LIN {X 0,Y 192.638,Z 331.481,A -85,B 0,C 180,E1 -21988.889,E2 -21988.889} C_VEL
LIN {X 0,Y 192.591,Z 331.489,A -85,B 0,C 180,E1 -21993.187,E2 -21993.187} C_VEL
LIN {X 0,Y 192.537,Z 331.501,A -85,B 0,C 180,E1 -21998.355,E2 -21998.355} C_VEL
LIN {X 0,Y 192.482,Z 331.497,A -85,B 0,C 180,E1 -22003.096,E2 -22003.096} C_VEL
LIN {X 0,Y 192.486,Z 331.508,A -85,B 0,C 180,E1 -22006.906,E2 -22006.906} C_VEL
LIN {X 0,Y 192.597,Z 331.632,A -85,B 0,C 180,E1 -22009.624,E2 -22009.624} C_VEL
LIN {X 0,Y 193.929,Z 336.776,A -85,B 0,C 180,E1 -22012.331,E2 -22012.331} C_VEL
LIN {X 0,Y 200.85,Z 352.206,A -85,B 0,C 180,E1 -22014.229,E2 -22014.229} C_VEL
LIN {X 0,Y 205.994,Z 365.473,A -85,B 0,C 180,E1 -22015.61,E2 -22015.61} C_VEL
LIN {X 0,Y 207.555,Z 370.626,A -85,B 0,C 180,E1 -22016.057,E2 -22016.057} C_VEL
LIN {X 0,Y 209.387,Z 387.344,A -85,B 0,C 180,E1 -22016.98,E2 -22016.98} C_VEL
LIN {X 0,Y 209.345,Z 391.227,A -85,B 0,C 180,E1 -22017.123,E2 -22017.123} C_VEL
LIN {X 0,Y 208.715,Z 395.103,A -85,B 0,C 180,E1 -22017.18,E2 -22017.18} C_VEL
LIN {X 0,Y 203.389,Z 412.296,A -85,B 0,C 180,E1 -22017.059,E2 -22017.059} C_VEL
LIN {X 0,Y 202.508,Z 418.198,A -85,B 0,C 180,E1 -22017.16,E2 -22017.16} C_VEL
LIN {X 0,Y 201.25,Z 446.446,A -85,B 0,C 180,E1 -22018.177,E2 -22018.177} C_VEL
LIN {X 0,Y 199.917,Z 460.229,A -85,B 0,C 180,E1 -22019.062,E2 -22019.062} C_VEL
LIN {X 0,Y 198.125,Z 472.398,A -85,B 0,C 180,E1 -22020.226,E2 -22020.226} C_VEL
LIN {X 0,Y 195.88,Z 485.013,A -85,B 0,C 180,E1 -22021.908,E2 -22021.908} C_VEL
LIN {X 0,Y 193.499,Z 496.249,A -85,B 0,C 180,E1 -22023.873,E2 -22023.873} C_VEL
LIN {X 0,Y 191.119,Z 506.332,A -85,B 0,C 180,E1 -22026.142,E2 -22026.142} C_VEL
LIN {X 0,Y 189.005,Z 515.48,A -85,B 0,C 180,E1 -22028.746,E2 -22028.746} C_VEL
LIN {X 0,Y 187.157,Z 523.008,A -85,B 0,C 180,E1 -22031.388,E2 -22031.388} C_VEL
LIN {X 0,Y 185.383,Z 530.39,A -85,B 0,C 180,E1 -22034.613,E2 -22034.613} C_VEL
LIN {X 0,Y 184.201,Z 536.3,A -85,B 0,C 180,E1 -22037.888,E2 -22037.888} C_VEL
LIN {X 0,Y 183.5,Z 540.938,A -85,B 0,C 180,E1 -22041.189,E2 -22041.189} C_VEL
LIN {X 0,Y 183.213,Z 543.376,A -85,B 0,C 180,E1 -22043.393,E2 -22043.393} C_VEL
LIN {X 0,Y 183.047,Z 546.146,A -85,B 0,C 180,E1 -22046.616,E2 -22046.616} C_VEL
LIN {X 0,Y 183.217,Z 548.062,A -85,B 0,C 180,E1 -22050.002,E2 -22050.002} C_VEL
LIN {X 0,Y 183.079,Z 549.003,A -85,B 0,C 180,E1 -22053.551,E2 -22053.551} C_VEL
LIN {X 0,Y 183.216,Z 548.977,A -85,B 0,C 180,E1 -22056.61,E2 -22056.61} C_VEL
LIN {X 0,Y 183.532,Z 548.51,A -85,B 0,C 180,E1 -22058.812,E2 -22058.812} C_VEL
LIN {X 0,Y 184.851,Z 546.339,A -85,B 0,C 180,E1 -22063.188,E2 -22063.188} C_VEL
LIN {X 0,Y 186.461,Z 543.652,A -85,B 0,C 180,E1 -22066.422,E2 -22066.422} C_VEL
LIN {X 0,Y 188.748,Z 539.973,A -85,B 0,C 180,E1 -22069.581,E2 -22069.581} C_VEL
LIN {X 0,Y 191.549,Z 535.205,A -85,B 0,C 180,E1 -22072.661,E2 -22072.661} C_VEL
LIN {X 0,Y 195.413,Z 528.093,A -85,B 0,C 180,E1 -22076.142,E2 -22076.142} C_VEL
LIN {X 0,Y 199.258,Z 520.373,A -85,B 0,C 180,E1 -22079.012,E2 -22079.012} C_VEL
LIN {X 0,Y 203.838,Z 510.725,A -85,B 0,C 180,E1 -22081.723,E2 -22081.723} C_VEL
LIN {X 0,Y 207.989,Z 500.784,A -85,B 0,C 180,E1 -22083.887,E2 -22083.887} C_VEL
LIN {X 0,Y 211.889,Z 489.576,A -85,B 0,C 180,E1 -22085.775,E2 -22085.775} C_VEL
LIN {X 0,Y 215.214,Z 478.603,A -85,B 0,C 180,E1 -22087.168,E2 -22087.168} C_VEL
LIN {X 0,Y 218.167,Z 466.461,A -85,B 0,C 180,E1 -22088.326,E2 -22088.326} C_VEL
LIN {X 0,Y 220.337,Z 454.664,A -85,B 0,C 180,E1 -22089.122,E2 -22089.122} C_VEL
LIN {X 0,Y 221.771,Z 441.816,A -85,B 0,C 180,E1 -22089.709,E2 -22089.709} C_VEL
LIN {X 0,Y 224.212,Z 400.799,A -85,B 0,C 180,E1 -22090.951,E2 -22090.951} C_VEL
LIN {X 0,Y 221.637,Z 393.948,A -85,B 0,C 180,E1 -22091.949,E2 -22091.949} C_VEL
LIN {X 0,Y 215.367,Z 380.157,A -85,B 0,C 180,E1 -22094.421,E2 -22094.421} C_VEL
LIN {X 0,Y 208.591,Z 367.511,A -85,B 0,C 180,E1 -22097.307,E2 -22097.307} C_VEL
LIN {X 0,Y 202.439,Z 357.412,A -85,B 0,C 180,E1 -22100.202,E2 -22100.202} C_VEL
LIN {X 0,Y 198.453,Z 351.457,A -85,B 0,C 180,E1 -22102.266,E2 -22102.266} C_VEL
LIN {X 0,Y 194.893,Z 346.176,A -85,B 0,C 180,E1 -22104.287,E2 -22104.287} C_VEL
LIN {X 0,Y 191.463,Z 341.379,A -85,B 0,C 180,E1 -22106.418,E2 -22106.418} C_VEL
LIN {X 0,Y 190.355,Z 339.981,A -85,B 0,C 180,E1 -22107.143,E2 -22107.143} C_VEL
LIN {X 0,Y 186.188,Z 334.613,A -85,B 0,C 180,E1 -22110.14,E2 -22110.14} C_VEL
LIN {X 0,Y 185.92,Z 333.953,A -85,B 0,C 180,E1 -22110.567,E2 -22110.567} C_VEL
LIN {X 0,Y 185.524,Z 332.37,A -85,B 0,C 180,E1 -22112.657,E2 -22112.657} C_VEL
LIN {X 0,Y 185.583,Z 332.358,A -85,B 0,C 180,E1 -22115.382,E2 -22115.382} C_VEL
LIN {X 0,Y 185.631,Z 332.362,A -85,B 0,C 180,E1 -22121.177,E2 -22121.177} C_VEL
LIN {X 0,Y 185.671,Z 332.35,A -85,B 0,C 180,E1 -22124.636,E2 -22124.636} C_VEL
LIN {X 0,Y 185.892,Z 332.325,A -85,B 0,C 180,E1 -22129.419,E2 -22129.419} C_VEL
LIN {X 0,Y 185.944,Z 332.316,A -85,B 0,C 180,E1 -22133.49,E2 -22133.49} C_VEL
LIN {X 0,Y 186.186,Z 332.285,A -85,B 0,C 180,E1 -22137.837,E2 -22137.837} C_VEL
LIN {X 0,Y 186.399,Z 332.249,A -85,B 0,C 180,E1 -22140,E2 -22140} C_VEL
LIN {X 0,Y 185.907,Z 332.313,A -85,B 0,C 180,E1 -22144.337,E2 -22144.337} C_VEL
LIN {X 0,Y 185.981,Z 332.306,A -85,B 0,C 180,E1 -22148.694,E2 -22148.694} C_VEL
LIN {X 0,Y 185.727,Z 332.338,A -85,B 0,C 180,E1 -22153.124,E2 -22153.124} C_VEL
LIN {X 0,Y 185.69,Z 332.458,A -85,B 0,C 180,E1 -22158.755,E2 -22158.755} C_VEL
LIN {X 0,Y 186.392,Z 334.808,A -85,B 0,C 180,E1 -22159.436,E2 -22159.436} C_VEL
LIN {X 0,Y 188.203,Z 337.049,A -85,B 0,C 180,E1 -22160.779,E2 -22160.779} C_VEL
LIN {X 0,Y 190.263,Z 338.408,A -85,B 0,C 180,E1 -22162.106,E2 -22162.106} C_VEL
LIN {X 0,Y 192.016,Z 341.447,A -85,B 0,C 180,E1 -22163.313,E2 -22163.313} C_VEL
LIN {X 0,Y 194.469,Z 343.734,A -85,B 0,C 180,E1 -22164.755,E2 -22164.755} C_VEL
LIN {X 0,Y 196.792,Z 347.187,A -85,B 0,C 180,E1 -22166.117,E2 -22166.117} C_VEL
LIN {X 0,Y 198.463,Z 348.976,A -85,B 0,C 180,E1 -22167.001,E2 -22167.001} C_VEL
LIN {X 0,Y 201.253,Z 352.699,A -85,B 0,C 180,E1 -22168.446,E2 -22168.446} C_VEL
LIN {X 0,Y 206.02,Z 359.299,A -85,B 0,C 180,E1 -22170.726,E2 -22170.726} C_VEL
LIN {X 0,Y 211.19,Z 366.859,A -85,B 0,C 180,E1 -22172.976,E2 -22172.976} C_VEL
LIN {X 0,Y 216.737,Z 376.683,A -85,B 0,C 180,E1 -22175.248,E2 -22175.248} C_VEL
LIN {X 0,Y 222.914,Z 389.306,A -85,B 0,C 180,E1 -22177.608,E2 -22177.608} C_VEL
LIN {X 0,Y 224.598,Z 393.07,A -85,B 0,C 180,E1 -22178.227,E2 -22178.227} C_VEL
LIN {X 0,Y 221.905,Z 436.193,A -85,B 0,C 180,E1 -22179.548,E2 -22179.548} C_VEL
LIN {X 0,Y 220.127,Z 449.537,A -85,B 0,C 180,E1 -22180.247,E2 -22180.247} C_VEL
LIN {X 0,Y 217.847,Z 461.771,A -85,B 0,C 180,E1 -22181.227,E2 -22181.227} C_VEL
LIN {X 0,Y 215.259,Z 472.394,A -85,B 0,C 180,E1 -22182.379,E2 -22182.379} C_VEL
LIN {X 0,Y 211.894,Z 483.788,A -85,B 0,C 180,E1 -22184.018,E2 -22184.018} C_VEL
LIN {X 0,Y 207.815,Z 495.071,A -85,B 0,C 180,E1 -22186.108,E2 -22186.108} C_VEL
LIN {X 0,Y 203.785,Z 504.611,A -85,B 0,C 180,E1 -22188.402,E2 -22188.402} C_VEL
LIN {X 0,Y 199.386,Z 513.782,A -85,B 0,C 180,E1 -22191.268,E2 -22191.268} C_VEL
LIN {X 0,Y 195.482,Z 521.122,A -85,B 0,C 180,E1 -22194.251,E2 -22194.251} C_VEL
LIN {X 0,Y 192.19,Z 526.777,A -85,B 0,C 180,E1 -22197.254,E2 -22197.254} C_VEL
LIN {X 0,Y 188.872,Z 532.063,A -85,B 0,C 180,E1 -22201.069,E2 -22201.069} C_VEL
LIN {X 0,Y 186.497,Z 535.594,A -85,B 0,C 180,E1 -22204.747,E2 -22204.747} C_VEL
LIN {X 0,Y 185.051,Z 537.448,A -85,B 0,C 180,E1 -22207.678,E2 -22207.678} C_VEL
LIN {X 0,Y 184.206,Z 538.371,A -85,B 0,C 180,E1 -22209.916,E2 -22209.916} C_VEL
LIN {X 0,Y 183.436,Z 538.951,A -85,B 0,C 180,E1 -22213.304,E2 -22213.304} C_VEL
LIN {X 0,Y 182.948,Z 538.61,A -85,B 0,C 180,E1 -22216.672,E2 -22216.672} C_VEL
LIN {X 0,Y 182.828,Z 537.889,A -85,B 0,C 180,E1 -22218.917,E2 -22218.917} C_VEL
LIN {X 0,Y 182.874,Z 536.746,A -85,B 0,C 180,E1 -22221.156,E2 -22221.156} C_VEL
LIN {X 0,Y 183.369,Z 533.537,A -85,B 0,C 180,E1 -22225.218,E2 -22225.218} C_VEL
LIN {X 0,Y 184.024,Z 529.31,A -85,B 0,C 180,E1 -22228.904,E2 -22228.904} C_VEL
LIN {X 0,Y 185.063,Z 524.327,A -85,B 0,C 180,E1 -22232.175,E2 -22232.175} C_VEL
LIN {X 0,Y 186.473,Z 518.077,A -85,B 0,C 180,E1 -22235.405,E2 -22235.405} C_VEL
LIN {X 0,Y 188.493,Z 510.24,A -85,B 0,C 180,E1 -22238.575,E2 -22238.575} C_VEL
LIN {X 0,Y 190.843,Z 500.485,A -85,B 0,C 180,E1 -22241.684,E2 -22241.684} C_VEL
LIN {X 0,Y 193.083,Z 491.441,A -85,B 0,C 180,E1 -22243.952,E2 -22243.952} C_VEL
LIN {X 0,Y 195.395,Z 481.62,A -85,B 0,C 180,E1 -22245.916,E2 -22245.916} C_VEL
LIN {X 0,Y 197.62,Z 469.256,A -85,B 0,C 180,E1 -22247.861,E2 -22247.861} C_VEL
LIN {X 0,Y 199.351,Z 457.162,A -85,B 0,C 180,E1 -22249.298,E2 -22249.298} C_VEL
LIN {X 0,Y 200.726,Z 444.557,A -85,B 0,C 180,E1 -22250.36,E2 -22250.36} C_VEL
LIN {X 0,Y 201.709,Z 431.047,A -85,B 0,C 180,E1 -22251.068,E2 -22251.068} C_VEL
LIN {X 0,Y 204.281,Z 372.696,A -85,B 0,C 180,E1 -22253.008,E2 -22253.008} C_VEL
LIN {X 0,Y 198.013,Z 356.135,A -85,B 0,C 180,E1 -22254.731,E2 -22254.731} C_VEL
LIN {X 0,Y 191.205,Z 342.963,A -85,B 0,C 180,E1 -22256.556,E2 -22256.556} C_VEL
LIN {X 0,Y 187.107,Z 335.978,A -85,B 0,C 180,E1 -22257.694,E2 -22257.694} C_VEL
LIN {X 0,Y 185.761,Z 333.349,A -85,B 0,C 180,E1 -22258.098,E2 -22258.098} C_VEL
LIN {X 0,Y 185.576,Z 332.366,A -85,B 0,C 180,E1 -22258.223,E2 -22258.223} C_VEL
LIN {X 0,Y 185.527,Z 332.372,A -85,B 0,C 180,E1 -22263.55,E2 -22263.55} C_VEL
LIN {X 0,Y 185.497,Z 332.379,A -85,B 0,C 180,E1 -22267.313,E2 -22267.313} C_VEL
LIN {X 0,Y 185.458,Z 332.373,A -85,B 0,C 180,E1 -22270.719,E2 -22270.719} C_VEL
LIN {X 0,Y 185.451,Z 332.373,A -85,B 0,C 180,E1 -22276.055,E2 -22276.055} C_VEL
LIN {X 0,Y 185.452,Z 332.381,A -85,B 0,C 180,E1 -22279.89,E2 -22279.89} C_VEL
LIN {X 0,Y 185.496,Z 332.369,A -85,B 0,C 180,E1 -22282.712,E2 -22282.712} C_VEL
LIN {X 0,Y 185.526,Z 332.371,A -85,B 0,C 180,E1 -22287.971,E2 -22287.971} C_VEL
LIN {X 0,Y 185.542,Z 332.369,A -85,B 0,C 180,E1 -22290.594,E2 -22290.594} C_VEL
LIN {X 0,Y 185.539,Z 332.352,A -85,B 0,C 180,E1 -22295.375,E2 -22295.375} C_VEL
LIN {X 0,Y 185.619,Z 332.36,A -85,B 0,C 180,E1 -22301.178,E2 -22301.178} C_VEL
LIN {X 0,Y 185.677,Z 332.344,A -85,B 0,C 180,E1 -22306.873,E2 -22306.873} C_VEL
LIN {X 0,Y 185.963,Z 332.318,A -85,B 0,C 180,E1 -22311.305,E2 -22311.305} C_VEL
LIN {X 0,Y 186.17,Z 332.283,A -85,B 0,C 180,E1 -22317.836,E2 -22317.836} C_VEL
LIN {X 0,Y 186.372,Z 332.268,A -85,B 0,C 180,E1 -22320,E2 -22320} C_VEL
LIN {X 0,Y 185.881,Z 332.311,A -85,B 0,C 180,E1 -22324.336,E2 -22324.336} C_VEL
LIN {X 0,Y 185.969,Z 332.312,A -85,B 0,C 180,E1 -22328.694,E2 -22328.694} C_VEL
LIN {X 0,Y 185.71,Z 332.344,A -85,B 0,C 180,E1 -22333.124,E2 -22333.124} C_VEL
LIN {X 0,Y 185.65,Z 332.349,A -85,B 0,C 180,E1 -22337.629,E2 -22337.629} C_VEL
LIN {X 0,Y 185.567,Z 332.365,A -85,B 0,C 180,E1 -22342.255,E2 -22342.255} C_VEL
LIN {X 0,Y 185.552,Z 332.369,A -85,B 0,C 180,E1 -22347.033,E2 -22347.033} C_VEL
LIN {X 0,Y 185.572,Z 332.364,A -85,B 0,C 180,E1 -22349.494,E2 -22349.494} C_VEL
LIN {X 0,Y 185.492,Z 332.377,A -85,B 0,C 180,E1 -22354.633,E2 -22354.633} C_VEL
LIN {X 0,Y 185.494,Z 332.374,A -85,B 0,C 180,E1 -22357.316,E2 -22357.316} C_VEL
LIN {X 0,Y 185.458,Z 332.375,A -85,B 0,C 180,E1 -22360.723,E2 -22360.723} C_VEL
LIN {X 0,Y 185.454,Z 332.382,A -85,B 0,C 180,E1 -22366.056,E2 -22366.056} C_VEL
LIN {X 0,Y 185.499,Z 332.529,A -85,B 0,C 180,E1 -22368.641,E2 -22368.641} C_VEL
LIN {X 0,Y 186.525,Z 336.356,A -85,B 0,C 180,E1 -22370.836,E2 -22370.836} C_VEL
LIN {X 0,Y 193.9,Z 352.127,A -85,B 0,C 180,E1 -22372.99,E2 -22372.99} C_VEL
LIN {X 0,Y 199.778,Z 367.06,A -85,B 0,C 180,E1 -22374.658,E2 -22374.658} C_VEL
LIN {X 0,Y 201.519,Z 372.667,A -85,B 0,C 180,E1 -22375.178,E2 -22375.178} C_VEL
LIN {X 0,Y 203.563,Z 393.383,A -85,B 0,C 180,E1 -22376.336,E2 -22376.336} C_VEL
LIN {X 0,Y 202.508,Z 418.198,A -85,B 0,C 180,E1 -22377.16,E2 -22377.16} C_VEL
LIN {X 0,Y 201.704,Z 424.041,A -85,B 0,C 180,E1 -22377.264,E2 -22377.264} C_VEL
LIN {X 0,Y 195.797,Z 442.985,A -85,B 0,C 180,E1 -22377.161,E2 -22377.161} C_VEL
LIN {X 0,Y 194.79,Z 448.778,A -85,B 0,C 180,E1 -22377.357,E2 -22377.357} C_VEL
LIN {X 0,Y 193.459,Z 461.067,A -85,B 0,C 180,E1 -22378.216,E2 -22378.216} C_VEL
LIN {X 0,Y 191.463,Z 473.919,A -85,B 0,C 180,E1 -22379.537,E2 -22379.537} C_VEL
LIN {X 0,Y 189.292,Z 485.383,A -85,B 0,C 180,E1 -22381.143,E2 -22381.143} C_VEL
LIN {X 0,Y 186.81,Z 496.491,A -85,B 0,C 180,E1 -22383.165,E2 -22383.165} C_VEL
LIN {X 0,Y 184.319,Z 506.582,A -85,B 0,C 180,E1 -22385.534,E2 -22385.534} C_VEL
LIN {X 0,Y 182.12,Z 515.677,A -85,B 0,C 180,E1 -22388.236,E2 -22388.236} C_VEL
LIN {X 0,Y 180.072,Z 523.741,A -85,B 0,C 180,E1 -22391.219,E2 -22391.219} C_VEL
LIN {X 0,Y 178.234,Z 530.943,A -85,B 0,C 180,E1 -22394.566,E2 -22394.566} C_VEL
LIN {X 0,Y 176.923,Z 537.493,A -85,B 0,C 180,E1 -22398.546,E2 -22398.546} C_VEL
LIN {X 0,Y 176.276,Z 541.802,A -85,B 0,C 180,E1 -22401.98,E2 -22401.98} C_VEL
LIN {X 0,Y 176.006,Z 545.02,A -85,B 0,C 180,E1 -22405.421,E2 -22405.421} C_VEL
LIN {X 0,Y 176.017,Z 546.614,A -85,B 0,C 180,E1 -22407.713,E2 -22407.713} C_VEL
LIN {X 0,Y 176.121,Z 547.793,A -85,B 0,C 180,E1 -22410.002,E2 -22410.002} C_VEL
LIN {X 0,Y 175.99,Z 548.712,A -85,B 0,C 180,E1 -22413.293,E2 -22413.293} C_VEL
LIN {X 0,Y 176.145,Z 548.791,A -85,B 0,C 180,E1 -22416.876,E2 -22416.876} C_VEL
LIN {X 0,Y 176.494,Z 548.36,A -85,B 0,C 180,E1 -22419.167,E2 -22419.167} C_VEL
LIN {X 0,Y 177.089,Z 547.51,A -85,B 0,C 180,E1 -22421.447,E2 -22421.447} C_VEL
LIN {X 0,Y 178.957,Z 544.608,A -85,B 0,C 180,E1 -22425.958,E2 -22425.958} C_VEL
LIN {X 0,Y 181.168,Z 541.319,A -85,B 0,C 180,E1 -22429.254,E2 -22429.254} C_VEL
LIN {X 0,Y 183.941,Z 536.988,A -85,B 0,C 180,E1 -22432.464,E2 -22432.464} C_VEL
LIN {X 0,Y 187.192,Z 531.603,A -85,B 0,C 180,E1 -22435.516,E2 -22435.516} C_VEL
LIN {X 0,Y 190.997,Z 524.661,A -85,B 0,C 180,E1 -22438.579,E2 -22438.579} C_VEL
LIN {X 0,Y 194.617,Z 517.703,A -85,B 0,C 180,E1 -22440.972,E2 -22440.972} C_VEL
LIN {X 0,Y 198.68,Z 509.341,A -85,B 0,C 180,E1 -22443.251,E2 -22443.251} C_VEL
LIN {X 0,Y 203.042,Z 499.05,A -85,B 0,C 180,E1 -22445.436,E2 -22445.436} C_VEL
LIN {X 0,Y 206.701,Z 488.898,A -85,B 0,C 180,E1 -22447.123,E2 -22447.123} C_VEL
LIN {X 0,Y 210.152,Z 477.81,A -85,B 0,C 180,E1 -22448.527,E2 -22448.527} C_VEL
LIN {X 0,Y 213.197,Z 465.472,A -85,B 0,C 180,E1 -22449.696,E2 -22449.696} C_VEL
LIN {X 0,Y 215.539,Z 452.357,A -85,B 0,C 180,E1 -22450.55,E2 -22450.55} C_VEL
LIN {X 0,Y 216.965,Z 438.806,A -85,B 0,C 180,E1 -22451.123,E2 -22451.123} C_VEL
LIN {X 0,Y 219.177,Z 402.734,A -85,B 0,C 180,E1 -22452.214,E2 -22452.214} C_VEL
LIN {X 0,Y 214.079,Z 390.468,A -85,B 0,C 180,E1 -22454.298,E2 -22454.298} C_VEL
LIN {X 0,Y 208.975,Z 379.906,A -85,B 0,C 180,E1 -22456.498,E2 -22456.498} C_VEL
LIN {X 0,Y 203.933,Z 370.682,A -85,B 0,C 180,E1 -22458.826,E2 -22458.826} C_VEL
LIN {X 0,Y 199.264,Z 362.827,A -85,B 0,C 180,E1 -22461.181,E2 -22461.181} C_VEL
LIN {X 0,Y 195.375,Z 356.854,A -85,B 0,C 180,E1 -22463.313,E2 -22463.313} C_VEL
LIN {X 0,Y 192.139,Z 351.892,A -85,B 0,C 180,E1 -22465.263,E2 -22465.263} C_VEL
LIN {X 0,Y 188.412,Z 346.551,A -85,B 0,C 180,E1 -22467.733,E2 -22467.733} C_VEL
LIN {X 0,Y 183.975,Z 340.613,A -85,B 0,C 180,E1 -22471.095,E2 -22471.095} C_VEL
LIN {X 0,Y 181.726,Z 338.38,A -85,B 0,C 180,E1 -22472.973,E2 -22472.973} C_VEL
LIN {X 0,Y 179.648,Z 336.3,A -85,B 0,C 180,E1 -22474.906,E2 -22474.906} C_VEL
LIN {X 0,Y 178.607,Z 333.868,A -85,B 0,C 180,E1 -22476.147,E2 -22476.147} C_VEL
LIN {X 0,Y 178.501,Z 333.248,A -85,B 0,C 180,E1 -22476.814,E2 -22476.814} C_VEL
LIN {X 0,Y 178.613,Z 333.232,A -85,B 0,C 180,E1 -22481.653,E2 -22481.653} C_VEL
LIN {X 0,Y 178.647,Z 333.22,A -85,B 0,C 180,E1 -22486.347,E2 -22486.347} C_VEL
LIN {X 0,Y 178.913,Z 333.183,A -85,B 0,C 180,E1 -22490.96,E2 -22490.96} C_VEL
LIN {X 0,Y 178.848,Z 333.189,A -85,B 0,C 180,E1 -22495.493,E2 -22495.493} C_VEL
LIN {X 0,Y 179.362,Z 333.126,A -85,B 0,C 180,E1 -22500,E2 -22500} C_VEL
LIN {X 0,Y 178.855,Z 333.19,A -85,B 0,C 180,E1 -22504.508,E2 -22504.508} C_VEL
LIN {X 0,Y 178.911,Z 333.185,A -85,B 0,C 180,E1 -22509.041,E2 -22509.041} C_VEL
LIN {X 0,Y 178.686,Z 333.326,A -85,B 0,C 180,E1 -22513.288,E2 -22513.288} C_VEL
LIN {X 0,Y 179.414,Z 335.699,A -85,B 0,C 180,E1 -22514.244,E2 -22514.244} C_VEL
LIN {X 0,Y 181.411,Z 338.026,A -85,B 0,C 180,E1 -22516.168,E2 -22516.168} C_VEL
LIN {X 0,Y 183.56,Z 339.35,A -85,B 0,C 180,E1 -22517.915,E2 -22517.915} C_VEL
LIN {X 0,Y 184.981,Z 342.119,A -85,B 0,C 180,E1 -22519.158,E2 -22519.158} C_VEL
LIN {X 0,Y 187.448,Z 344.411,A -85,B 0,C 180,E1 -22520.936,E2 -22520.936} C_VEL
LIN {X 0,Y 188.244,Z 345.296,A -85,B 0,C 180,E1 -22521.489,E2 -22521.489} C_VEL
LIN {X 0,Y 190.555,Z 348.614,A -85,B 0,C 180,E1 -22523.071,E2 -22523.071} C_VEL
LIN {X 0,Y 192.224,Z 350.358,A -85,B 0,C 180,E1 -22524.094,E2 -22524.094} C_VEL
LIN {X 0,Y 195.069,Z 354.109,A -85,B 0,C 180,E1 -22525.778,E2 -22525.778} C_VEL
LIN {X 0,Y 199.775,Z 360.495,A -85,B 0,C 180,E1 -22528.314,E2 -22528.314} C_VEL
LIN {X 0,Y 204.677,Z 367.388,A -85,B 0,C 180,E1 -22530.69,E2 -22530.69} C_VEL
LIN {X 0,Y 209.07,Z 374.425,A -85,B 0,C 180,E1 -22532.664,E2 -22532.664} C_VEL
LIN {X 0,Y 214.568,Z 384.816,A -85,B 0,C 180,E1 -22534.994,E2 -22534.994} C_VEL
LIN {X 0,Y 219.591,Z 395.691,A -85,B 0,C 180,E1 -22536.995,E2 -22536.995} C_VEL
LIN {X 0,Y 216.925,Z 435.881,A -85,B 0,C 180,E1 -22538.218,E2 -22538.218} C_VEL
LIN {X 0,Y 215.103,Z 449.326,A -85,B 0,C 180,E1 -22538.919,E2 -22538.919} C_VEL
LIN {X 0,Y 212.612,Z 462.237,A -85,B 0,C 180,E1 -22539.96,E2 -22539.96} C_VEL
LIN {X 0,Y 209.929,Z 472.795,A -85,B 0,C 180,E1 -22541.125,E2 -22541.125} C_VEL
LIN {X 0,Y 206.259,Z 484.606,A -85,B 0,C 180,E1 -22542.86,E2 -22542.86} C_VEL
LIN {X 0,Y 202.175,Z 495.399,A -85,B 0,C 180,E1 -22544.904,E2 -22544.904} C_VEL
LIN {X 0,Y 198.383,Z 504.062,A -85,B 0,C 180,E1 -22547.002,E2 -22547.002} C_VEL
LIN {X 0,Y 193.724,Z 513.37,A -85,B 0,C 180,E1 -22549.912,E2 -22549.912} C_VEL
LIN {X 0,Y 189.546,Z 520.819,A -85,B 0,C 180,E1 -22552.948,E2 -22552.948} C_VEL
LIN {X 0,Y 185.755,Z 527.083,A -85,B 0,C 180,E1 -22556.343,E2 -22556.343} C_VEL
LIN {X 0,Y 182.465,Z 531.979,A -85,B 0,C 180,E1 -22559.951,E2 -22559.951} C_VEL
LIN {X 0,Y 179.673,Z 535.88,A -85,B 0,C 180,E1 -22564.115,E2 -22564.115} C_VEL
LIN {X 0,Y 178.293,Z 537.522,A -85,B 0,C 180,E1 -22566.784,E2 -22566.784} C_VEL
LIN {X 0,Y 176.699,Z 539.042,A -85,B 0,C 180,E1 -22571.445,E2 -22571.445} C_VEL
LIN {X 0,Y 176.259,Z 539.161,A -85,B 0,C 180,E1 -22573.791,E2 -22573.791} C_VEL
LIN {X 0,Y 175.92,Z 538.867,A -85,B 0,C 180,E1 -22576.13,E2 -22576.13} C_VEL
LIN {X 0,Y 175.732,Z 538.183,A -85,B 0,C 180,E1 -22578.464,E2 -22578.464} C_VEL
LIN {X 0,Y 175.754,Z 537.102,A -85,B 0,C 180,E1 -22580.794,E2 -22580.794} C_VEL
LIN {X 0,Y 175.938,Z 535.564,A -85,B 0,C 180,E1 -22583.116,E2 -22583.116} C_VEL
LIN {X 0,Y 176.491,Z 532.471,A -85,B 0,C 180,E1 -22586.574,E2 -22586.574} C_VEL
LIN {X 0,Y 177.168,Z 528.341,A -85,B 0,C 180,E1 -22589.998,E2 -22589.998} C_VEL
LIN {X 0,Y 178.65,Z 522.021,A -85,B 0,C 180,E1 -22593.946,E2 -22593.946} C_VEL
LIN {X 0,Y 180.402,Z 515.151,A -85,B 0,C 180,E1 -22597.272,E2 -22597.272} C_VEL
LIN {X 0,Y 182.638,Z 506.556,A -85,B 0,C 180,E1 -22600.53,E2 -22600.53} C_VEL
LIN {X 0,Y 184.88,Z 497.741,A -85,B 0,C 180,E1 -22603.182,E2 -22603.182} C_VEL
LIN {X 0,Y 187.447,Z 488.018,A -85,B 0,C 180,E1 -22605.492,E2 -22605.492} C_VEL
LIN {X 0,Y 189.745,Z 477.412,A -85,B 0,C 180,E1 -22607.512,E2 -22607.512} C_VEL
LIN {X 0,Y 191.831,Z 465.59,A -85,B 0,C 180,E1 -22609.25,E2 -22609.25} C_VEL
LIN {X 0,Y 193.501,Z 453.33,A -85,B 0,C 180,E1 -22610.599,E2 -22610.599} C_VEL
LIN {X 0,Y 194.819,Z 440.33,A -85,B 0,C 180,E1 -22611.591,E2 -22611.591} C_VEL
LIN {X 0,Y 195.722,Z 426.06,A -85,B 0,C 180,E1 -22612.211,E2 -22612.211} C_VEL
LIN {X 0,Y 198.024,Z 374.257,A -85,B 0,C 180,E1 -22613.975,E2 -22613.975} C_VEL
LIN {X 0,Y 192.432,Z 359.438,A -85,B 0,C 180,E1 -22615.6,E2 -22615.6} C_VEL
LIN {X 0,Y 186.083,Z 347.086,A -85,B 0,C 180,E1 -22617.398,E2 -22617.398} C_VEL
LIN {X 0,Y 180.27,Z 337.107,A -85,B 0,C 180,E1 -22619.128,E2 -22619.128} C_VEL
LIN {X 0,Y 178.831,Z 334.65,A -85,B 0,C 180,E1 -22619.578,E2 -22619.578} C_VEL
LIN {X 0,Y 178.491,Z 333.249,A -85,B 0,C 180,E1 -22619.754,E2 -22619.754} C_VEL
LIN {X 0,Y 178.481,Z 333.251,A -85,B 0,C 180,E1 -22624.216,E2 -22624.216} C_VEL
LIN {X 0,Y 178.384,Z 333.261,A -85,B 0,C 180,E1 -22629.075,E2 -22629.075} C_VEL
LIN {X 0,Y 178.39,Z 333.258,A -85,B 0,C 180,E1 -22632.045,E2 -22632.045} C_VEL
LIN {X 0,Y 178.388,Z 333.258,A -85,B 0,C 180,E1 -22635.163,E2 -22635.163} C_VEL
LIN {X 0,Y 178.393,Z 333.251,A -85,B 0,C 180,E1 -22638.46,E2 -22638.46} C_VEL
LIN {X 0,Y 178.414,Z 333.243,A -85,B 0,C 180,E1 -22643.78,E2 -22643.78} C_VEL
LIN {X 0,Y 178.479,Z 333.239,A -85,B 0,C 180,E1 -22646.544,E2 -22646.544} C_VEL
LIN {X 0,Y 178.433,Z 333.247,A -85,B 0,C 180,E1 -22651.793,E2 -22651.793} C_VEL
LIN {X 0,Y 178.458,Z 333.247,A -85,B 0,C 180,E1 -22656.807,E2 -22656.807} C_VEL
LIN {X 0,Y 178.599,Z 333.229,A -85,B 0,C 180,E1 -22661.65,E2 -22661.65} C_VEL
LIN {X 0,Y 178.608,Z 333.217,A -85,B 0,C 180,E1 -22666.343,E2 -22666.343} C_VEL
LIN {X 0,Y 178.894,Z 333.198,A -85,B 0,C 180,E1 -22670.958,E2 -22670.958} C_VEL
LIN {X 0,Y 179.117,Z 333.161,A -85,B 0,C 180,E1 -22677.751,E2 -22677.751} C_VEL
LIN {X 0,Y 179.338,Z 333.144,A -85,B 0,C 180,E1 -22680,E2 -22680} C_VEL
LIN {X 0,Y 178.829,Z 333.187,A -85,B 0,C 180,E1 -22684.508,E2 -22684.508} C_VEL
LIN {X 0,Y 178.899,Z 333.196,A -85,B 0,C 180,E1 -22689.04,E2 -22689.04} C_VEL
LIN {X 0,Y 178.637,Z 333.222,A -85,B 0,C 180,E1 -22693.653,E2 -22693.653} C_VEL
LIN {X 0,Y 178.584,Z 333.238,A -85,B 0,C 180,E1 -22699.186,E2 -22699.186} C_VEL
LIN {X 0,Y 178.514,Z 333.246,A -85,B 0,C 180,E1 -22705.115,E2 -22705.115} C_VEL
LIN {X 0,Y 178.516,Z 333.246,A -85,B 0,C 180,E1 -22709.994,E2 -22709.994} C_VEL
LIN {X 0,Y 178.478,Z 333.25,A -85,B 0,C 180,E1 -22714.219,E2 -22714.219} C_VEL
LIN {X 0,Y 178.383,Z 333.265,A -85,B 0,C 180,E1 -22719.077,E2 -22719.077} C_VEL
LIN {X 0,Y 178.39,Z 333.247,A -85,B 0,C 180,E1 -22722.047,E2 -22722.047} C_VEL
LIN {X 0,Y 178.436,Z 333.385,A -85,B 0,C 180,E1 -22727.552,E2 -22727.552} C_VEL
LIN {X 0,Y 179.219,Z 336.344,A -85,B 0,C 180,E1 -22729.229,E2 -22729.229} C_VEL
LIN {X 0,Y 185.613,Z 349.24,A -85,B 0,C 180,E1 -22731.238,E2 -22731.238} C_VEL
LIN {X 0,Y 191.601,Z 363.384,A -85,B 0,C 180,E1 -22733.05,E2 -22733.05} C_VEL
LIN {X 0,Y 195.466,Z 374.241,A -85,B 0,C 180,E1 -22734.215,E2 -22734.215} C_VEL
LIN {X 0,Y 197.345,Z 393.527,A -85,B 0,C 180,E1 -22735.342,E2 -22735.342} C_VEL
LIN {X 0,Y 195.021,Z 445.761,A -85,B 0,C 180,E1 -22737.199,E2 -22737.199} C_VEL
LIN {X 0,Y 194.79,Z 448.778,A -85,B 0,C 180,E1 -22737.357,E2 -22737.357} C_VEL
LIN {X 0,Y 193.646,Z 454.526,A -85,B 0,C 180,E1 -22737.603,E2 -22737.603} C_VEL
LIN {X 0,Y 189.956,Z 463.679,A -85,B 0,C 180,E1 -22737.942,E2 -22737.942} C_VEL
LIN {X 0,Y 185.957,Z 472.567,A -85,B 0,C 180,E1 -22738.514,E2 -22738.514} C_VEL
LIN {X 0,Y 184.344,Z 477.899,A -85,B 0,C 180,E1 -22739.129,E2 -22739.129} C_VEL
LIN {X 0,Y 181.754,Z 490.143,A -85,B 0,C 180,E1 -22741.098,E2 -22741.098} C_VEL
LIN {X 0,Y 179.193,Z 500.26,A -85,B 0,C 180,E1 -22743.192,E2 -22743.192} C_VEL
LIN {X 0,Y 176.667,Z 510.477,A -85,B 0,C 180,E1 -22745.938,E2 -22745.938} C_VEL
LIN {X 0,Y 174.574,Z 518.818,A -85,B 0,C 180,E1 -22748.759,E2 -22748.759} C_VEL
LIN {X 0,Y 172.299,Z 526.95,A -85,B 0,C 180,E1 -22752.188,E2 -22752.188} C_VEL
LIN {X 0,Y 170.605,Z 533.47,A -85,B 0,C 180,E1 -22755.692,E2 -22755.692} C_VEL
LIN {X 0,Y 169.659,Z 538.641,A -85,B 0,C 180,E1 -22759.259,E2 -22759.259} C_VEL
LIN {X 0,Y 169.093,Z 542.633,A -85,B 0,C 180,E1 -22762.839,E2 -22762.839} C_VEL
LIN {X 0,Y 168.891,Z 545.971,A -85,B 0,C 180,E1 -22767.08,E2 -22767.08} C_VEL
LIN {X 0,Y 169.027,Z 547.511,A -85,B 0,C 180,E1 -22770.002,E2 -22770.002} C_VEL
LIN {X 0,Y 168.891,Z 548.378,A -85,B 0,C 180,E1 -22772.923,E2 -22772.923} C_VEL
LIN {X 0,Y 169.097,Z 548.605,A -85,B 0,C 180,E1 -22777.164,E2 -22777.164} C_VEL
LIN {X 0,Y 170.113,Z 547.401,A -85,B 0,C 180,E1 -22781.923,E2 -22781.923} C_VEL
LIN {X 0,Y 172.112,Z 544.555,A -85,B 0,C 180,E1 -22786.611,E2 -22786.611} C_VEL
LIN {X 0,Y 174.471,Z 541.326,A -85,B 0,C 180,E1 -22790.024,E2 -22790.024} C_VEL
LIN {X 0,Y 177.391,Z 537.056,A -85,B 0,C 180,E1 -22793.342,E2 -22793.342} C_VEL
LIN {X 0,Y 181.187,Z 531.041,A -85,B 0,C 180,E1 -22796.857,E2 -22796.857} C_VEL
LIN {X 0,Y 185.516,Z 523.611,A -85,B 0,C 180,E1 -22800.131,E2 -22800.131} C_VEL
LIN {X 0,Y 190.227,Z 514.869,A -85,B 0,C 180,E1 -22803.022,E2 -22803.022} C_VEL
LIN {X 0,Y 194.58,Z 505.931,A -85,B 0,C 180,E1 -22805.305,E2 -22805.305} C_VEL
LIN {X 0,Y 198.699,Z 496.128,A -85,B 0,C 180,E1 -22807.281,E2 -22807.281} C_VEL
LIN {X 0,Y 202.631,Z 485.309,A -85,B 0,C 180,E1 -22808.951,E2 -22808.951} C_VEL
LIN {X 0,Y 206.243,Z 473.197,A -85,B 0,C 180,E1 -22810.351,E2 -22810.351} C_VEL
LIN {X 0,Y 209.142,Z 460.546,A -85,B 0,C 180,E1 -22811.422,E2 -22811.422} C_VEL
LIN {X 0,Y 211.155,Z 448.089,A -85,B 0,C 180,E1 -22812.131,E2 -22812.131} C_VEL
LIN {X 0,Y 212.568,Z 431.302,A -85,B 0,C 180,E1 -22812.719,E2 -22812.719} C_VEL
LIN {X 0,Y 214.233,Z 405.066,A -85,B 0,C 180,E1 -22813.522,E2 -22813.522} C_VEL
LIN {X 0,Y 208.846,Z 392.125,A -85,B 0,C 180,E1 -22815.885,E2 -22815.885} C_VEL
LIN {X 0,Y 203.558,Z 381.361,A -85,B 0,C 180,E1 -22818.347,E2 -22818.347} C_VEL
LIN {X 0,Y 198.497,Z 372.194,A -85,B 0,C 180,E1 -22820.912,E2 -22820.912} C_VEL
LIN {X 0,Y 195.302,Z 366.865,A -85,B 0,C 180,E1 -22822.667,E2 -22822.667} C_VEL
LIN {X 0,Y 192.472,Z 362.37,A -85,B 0,C 180,E1 -22824.332,E2 -22824.332} C_VEL
LIN {X 0,Y 189.629,Z 357.883,A -85,B 0,C 180,E1 -22826.146,E2 -22826.146} C_VEL
LIN {X 0,Y 185.942,Z 352.541,A -85,B 0,C 180,E1 -22828.727,E2 -22828.727} C_VEL
LIN {X 0,Y 181.364,Z 346.262,A -85,B 0,C 180,E1 -22832.446,E2 -22832.446} C_VEL
LIN {X 0,Y 178.038,Z 342.903,A -85,B 0,C 180,E1 -22835.568,E2 -22835.568} C_VEL
LIN {X 0,Y 176.725,Z 340.115,A -85,B 0,C 180,E1 -22837.186,E2 -22837.186} C_VEL
LIN {X 0,Y 173.842,Z 338.555,A -85,B 0,C 180,E1 -22840.718,E2 -22840.718} C_VEL
LIN {X 0,Y 172.06,Z 335.991,A -85,B 0,C 180,E1 -22843.844,E2 -22843.844} C_VEL
LIN {X 0,Y 171.544,Z 334.115,A -85,B 0,C 180,E1 -22845.316,E2 -22845.316} C_VEL
LIN {X 0,Y 171.85,Z 334.065,A -85,B 0,C 180,E1 -22850.585,E2 -22850.585} C_VEL
LIN {X 0,Y 171.798,Z 334.068,A -85,B 0,C 180,E1 -22855.307,E2 -22855.307} C_VEL
LIN {X 0,Y 172.325,Z 334.002,A -85,B 0,C 180,E1 -22860,E2 -22860} C_VEL
LIN {X 0,Y 171.822,Z 334.222,A -85,B 0,C 180,E1 -22864.766,E2 -22864.766} C_VEL
LIN {X 0,Y 172.458,Z 336.206,A -85,B 0,C 180,E1 -22866.288,E2 -22866.288} C_VEL
LIN {X 0,Y 174.454,Z 338.749,A -85,B 0,C 180,E1 -22869.517,E2 -22869.517} C_VEL
LIN {X 0,Y 176.991,Z 340.364,A -85,B 0,C 180,E1 -22872.542,E2 -22872.542} C_VEL
LIN {X 0,Y 178.173,Z 342.915,A -85,B 0,C 180,E1 -22873.981,E2 -22873.981} C_VEL
LIN {X 0,Y 180.4,Z 345.164,A -85,B 0,C 180,E1 -22876.116,E2 -22876.116} C_VEL
LIN {X 0,Y 181.641,Z 345.99,A -85,B 0,C 180,E1 -22877.16,E2 -22877.16} C_VEL
LIN {X 0,Y 183.605,Z 349.275,A -85,B 0,C 180,E1 -22878.881,E2 -22878.881} C_VEL
LIN {X 0,Y 186.033,Z 351.587,A -85,B 0,C 180,E1 -22880.671,E2 -22880.671} C_VEL
LIN {X 0,Y 188.554,Z 355.119,A -85,B 0,C 180,E1 -22882.461,E2 -22882.461} C_VEL
LIN {X 0,Y 190.044,Z 356.862,A -85,B 0,C 180,E1 -22883.425,E2 -22883.425} C_VEL
LIN {X 0,Y 192.936,Z 360.589,A -85,B 0,C 180,E1 -22885.198,E2 -22885.198} C_VEL
LIN {X 0,Y 199.557,Z 369.991,A -85,B 0,C 180,E1 -22888.82,E2 -22888.82} C_VEL
LIN {X 0,Y 205.215,Z 378.841,A -85,B 0,C 180,E1 -22891.546,E2 -22891.546} C_VEL
LIN {X 0,Y 210.736,Z 389.571,A -85,B 0,C 180,E1 -22894.027,E2 -22894.027} C_VEL
LIN {X 0,Y 214.59,Z 398.054,A -85,B 0,C 180,E1 -22895.664,E2 -22895.664} C_VEL
LIN {X 0,Y 211.953,Z 436.63,A -85,B 0,C 180,E1 -22896.874,E2 -22896.874} C_VEL
LIN {X 0,Y 210.065,Z 449.895,A -85,B 0,C 180,E1 -22897.579,E2 -22897.579} C_VEL
LIN {X 0,Y 207.49,Z 462.696,A -85,B 0,C 180,E1 -22898.631,E2 -22898.631} C_VEL
LIN {X 0,Y 204.703,Z 473.193,A -85,B 0,C 180,E1 -22899.807,E2 -22899.807} C_VEL
LIN {X 0,Y 200.98,Z 484.68,A -85,B 0,C 180,E1 -22901.511,E2 -22901.511} C_VEL
LIN {X 0,Y 196.631,Z 495.728,A -85,B 0,C 180,E1 -22903.631,E2 -22903.631} C_VEL
LIN {X 0,Y 192.24,Z 505.206,A -85,B 0,C 180,E1 -22906.002,E2 -22906.002} C_VEL
LIN {X 0,Y 188.204,Z 512.923,A -85,B 0,C 180,E1 -22908.464,E2 -22908.464} C_VEL
LIN {X 0,Y 183.736,Z 520.514,A -85,B 0,C 180,E1 -22911.568,E2 -22911.568} C_VEL
LIN {X 0,Y 180.542,Z 525.617,A -85,B 0,C 180,E1 -22914.272,E2 -22914.272} C_VEL
LIN {X 0,Y 177.155,Z 530.525,A -85,B 0,C 180,E1 -22917.616,E2 -22917.616} C_VEL
LIN {X 0,Y 174.385,Z 534.259,A -85,B 0,C 180,E1 -22921.076,E2 -22921.076} C_VEL
LIN {X 0,Y 172.87,Z 536.17,A -85,B 0,C 180,E1 -22923.434,E2 -22923.434} C_VEL
LIN {X 0,Y 171.591,Z 537.598,A -85,B 0,C 180,E1 -22925.82,E2 -22925.82} C_VEL
LIN {X 0,Y 169.789,Z 539.191,A -85,B 0,C 180,E1 -22930.66,E2 -22930.66} C_VEL
LIN {X 0,Y 169.261,Z 539.38,A -85,B 0,C 180,E1 -22933.101,E2 -22933.101} C_VEL
LIN {X 0,Y 168.877,Z 539.124,A -85,B 0,C 180,E1 -22935.539,E2 -22935.539} C_VEL
LIN {X 0,Y 168.654,Z 537.433,A -85,B 0,C 180,E1 -22940.403,E2 -22940.403} C_VEL
LIN {X 0,Y 168.823,Z 535.966,A -85,B 0,C 180,E1 -22942.824,E2 -22942.824} C_VEL
LIN {X 0,Y 169.297,Z 533.267,A -85,B 0,C 180,E1 -22946.096,E2 -22946.096} C_VEL
LIN {X 0,Y 170.06,Z 528.901,A -85,B 0,C 180,E1 -22949.998,E2 -22949.998} C_VEL
LIN {X 0,Y 171.547,Z 522.672,A -85,B 0,C 180,E1 -22954.11,E2 -22954.11} C_VEL
LIN {X 0,Y 173.369,Z 515.899,A -85,B 0,C 180,E1 -22957.569,E2 -22957.569} C_VEL
LIN {X 0,Y 175.697,Z 507.476,A -85,B 0,C 180,E1 -22960.951,E2 -22960.951} C_VEL
LIN {X 0,Y 177.986,Z 498.807,A -85,B 0,C 180,E1 -22963.703,E2 -22963.703} C_VEL
LIN {X 0,Y 180.645,Z 489.256,A -85,B 0,C 180,E1 -22966.091,E2 -22966.091} C_VEL
LIN {X 0,Y 183.046,Z 478.867,A -85,B 0,C 180,E1 -22968.175,E2 -22968.175} C_VEL
LIN {X 0,Y 185.207,Z 467.5,A -85,B 0,C 180,E1 -22969.968,E2 -22969.968} C_VEL
LIN {X 0,Y 186.932,Z 455.811,A -85,B 0,C 180,E1 -22971.357,E2 -22971.357} C_VEL
LIN {X 0,Y 188.416,Z 442.42,A -85,B 0,C 180,E1 -22972.47,E2 -22972.47} C_VEL
LIN {X 0,Y 189.351,Z 429.717,A -85,B 0,C 180,E1 -22973.113,E2 -22973.113} C_VEL
LIN {X 0,Y 191.862,Z 375.924,A -85,B 0,C 180,E1 -22974.991,E2 -22974.991} C_VEL
LIN {X 0,Y 186.796,Z 362.46,A -85,B 0,C 180,E1 -22976.553,E2 -22976.553} C_VEL
LIN {X 0,Y 179.583,Z 348.533,A -85,B 0,C 180,E1 -22978.731,E2 -22978.731} C_VEL
LIN {X 0,Y 174.862,Z 340.753,A -85,B 0,C 180,E1 -22980.217,E2 -22980.217} C_VEL
LIN {X 0,Y 173.327,Z 338.139,A -85,B 0,C 180,E1 -22980.727,E2 -22980.727} C_VEL
LIN {X 0,Y 171.776,Z 335.673,A -85,B 0,C 180,E1 -22981.247,E2 -22981.247} C_VEL
LIN {X 0,Y 171.394,Z 334.134,A -85,B 0,C 180,E1 -22981.507,E2 -22981.507} C_VEL
LIN {X 0,Y 171.39,Z 334.134,A -85,B 0,C 180,E1 -22985.033,E2 -22985.033} C_VEL
LIN {X 0,Y 171.34,Z 334.14,A -85,B 0,C 180,E1 -22988.799,E2 -22988.799} C_VEL
LIN {X 0,Y 171.315,Z 334.145,A -85,B 0,C 180,E1 -22994.216,E2 -22994.216} C_VEL
LIN {X 0,Y 171.326,Z 334.134,A -85,B 0,C 180,E1 -22998.978,E2 -22998.978} C_VEL
LIN {X 0,Y 171.356,Z 334.135,A -85,B 0,C 180,E1 -23002.032,E2 -23002.032} C_VEL
LIN {X 0,Y 171.393,Z 334.112,A -85,B 0,C 180,E1 -23005.091,E2 -23005.091} C_VEL
LIN {X 0,Y 171.402,Z 334.13,A -85,B 0,C 180,E1 -23010.525,E2 -23010.525} C_VEL
LIN {X 0,Y 171.398,Z 334.115,A -85,B 0,C 180,E1 -23015.792,E2 -23015.792} C_VEL
LIN {X 0,Y 171.502,Z 334.119,A -85,B 0,C 180,E1 -23020.862,E2 -23020.862} C_VEL
LIN {X 0,Y 171.527,Z 334.093,A -85,B 0,C 180,E1 -23025.768,E2 -23025.768} C_VEL
LIN {X 0,Y 171.834,Z 334.078,A -85,B 0,C 180,E1 -23030.584,E2 -23030.584} C_VEL
LIN {X 0,Y 171.775,Z 334.058,A -85,B 0,C 180,E1 -23035.306,E2 -23035.306} C_VEL
LIN {X 0,Y 172.302,Z 334.02,A -85,B 0,C 180,E1 -23040,E2 -23040} C_VEL
LIN {X 0,Y 171.779,Z 334.063,A -85,B 0,C 180,E1 -23044.693,E2 -23044.693} C_VEL
LIN {X 0,Y 171.838,Z 334.078,A -85,B 0,C 180,E1 -23049.415,E2 -23049.415} C_VEL
LIN {X 0,Y 171.551,Z 334.097,A -85,B 0,C 180,E1 -23054.229,E2 -23054.229} C_VEL
LIN {X 0,Y 171.509,Z 334.121,A -85,B 0,C 180,E1 -23059.534,E2 -23059.534} C_VEL
LIN {X 0,Y 171.452,Z 334.128,A -85,B 0,C 180,E1 -23065.609,E2 -23065.609} C_VEL
LIN {X 0,Y 171.434,Z 334.128,A -85,B 0,C 180,E1 -23070.586,E2 -23070.586} C_VEL
LIN {X 0,Y 171.386,Z 334.135,A -85,B 0,C 180,E1 -23075.036,E2 -23075.036} C_VEL
LIN {X 0,Y 171.338,Z 334.142,A -85,B 0,C 180,E1 -23078.803,E2 -23078.803} C_VEL
LIN {X 0,Y 171.315,Z 334.142,A -85,B 0,C 180,E1 -23084.219,E2 -23084.219} C_VEL
LIN {X 0,Y 171.4,Z 334.168,A -85,B 0,C 180,E1 -23086.322,E2 -23086.322} C_VEL
LIN {X 0,Y 171.825,Z 335.948,A -85,B 0,C 180,E1 -23087.411,E2 -23087.411} C_VEL
LIN {X 0,Y 173.908,Z 339.999,A -85,B 0,C 180,E1 -23088.143,E2 -23088.143} C_VEL
LIN {X 0,Y 180.145,Z 352.4,A -85,B 0,C 180,E1 -23090.215,E2 -23090.215} C_VEL
LIN {X 0,Y 186.575,Z 367.896,A -85,B 0,C 180,E1 -23092.282,E2 -23092.282} C_VEL
LIN {X 0,Y 189.484,Z 376.311,A -85,B 0,C 180,E1 -23093.219,E2 -23093.219} C_VEL
LIN {X 0,Y 191.182,Z 394.77,A -85,B 0,C 180,E1 -23094.334,E2 -23094.334} C_VEL
LIN {X 0,Y 188.851,Z 444.931,A -85,B 0,C 180,E1 -23096.15,E2 -23096.15} C_VEL
LIN {X 0,Y 187.507,Z 458.148,A -85,B 0,C 180,E1 -23097.002,E2 -23097.002} C_VEL
LIN {X 0,Y 185.72,Z 470.3,A -85,B 0,C 180,E1 -23098.171,E2 -23098.171} C_VEL
LIN {X 0,Y 184.344,Z 477.899,A -85,B 0,C 180,E1 -23099.129,E2 -23099.129} C_VEL
LIN {X 0,Y 182.614,Z 483.232,A -85,B 0,C 180,E1 -23099.82,E2 -23099.82} C_VEL
LIN {X 0,Y 177.983,Z 491.452,A -85,B 0,C 180,E1 -23100.865,E2 -23100.865} C_VEL
LIN {X 0,Y 173.353,Z 499.194,A -85,B 0,C 180,E1 -23102.168,E2 -23102.168} C_VEL
LIN {X 0,Y 171.649,Z 503.736,A -85,B 0,C 180,E1 -23103.244,E2 -23103.244} C_VEL
LIN {X 0,Y 169.279,Z 512.878,A -85,B 0,C 180,E1 -23105.976,E2 -23105.976} C_VEL
LIN {X 0,Y 167.005,Z 521.079,A -85,B 0,C 180,E1 -23109.043,E2 -23109.043} C_VEL
LIN {X 0,Y 164.875,Z 528.7,A -85,B 0,C 180,E1 -23112.641,E2 -23112.641} C_VEL
LIN {X 0,Y 163.285,Z 534.812,A -85,B 0,C 180,E1 -23116.309,E2 -23116.309} C_VEL
LIN {X 0,Y 162.391,Z 539.646,A -85,B 0,C 180,E1 -23120.033,E2 -23120.033} C_VEL
LIN {X 0,Y 161.894,Z 543.331,A -85,B 0,C 180,E1 -23123.771,E2 -23123.771} C_VEL
LIN {X 0,Y 161.836,Z 545.981,A -85,B 0,C 180,E1 -23127.513,E2 -23127.513} C_VEL
LIN {X 0,Y 161.937,Z 547.22,A -85,B 0,C 180,E1 -23130.002,E2 -23130.002} C_VEL
LIN {X 0,Y 161.812,Z 548.06,A -85,B 0,C 180,E1 -23132.617,E2 -23132.617} C_VEL
LIN {X 0,Y 161.85,Z 548.419,A -85,B 0,C 180,E1 -23134.984,E2 -23134.984} C_VEL
LIN {X 0,Y 162.453,Z 548.04,A -85,B 0,C 180,E1 -23139.967,E2 -23139.967} C_VEL
LIN {X 0,Y 163.157,Z 547.283,A -85,B 0,C 180,E1 -23142.439,E2 -23142.439} C_VEL
LIN {X 0,Y 164.109,Z 546.097,A -85,B 0,C 180,E1 -23144.891,E2 -23144.891} C_VEL
LIN {X 0,Y 165.293,Z 544.504,A -85,B 0,C 180,E1 -23147.317,E2 -23147.317} C_VEL
LIN {X 0,Y 167.81,Z 541.333,A -85,B 0,C 180,E1 -23150.855,E2 -23150.855} C_VEL
LIN {X 0,Y 170.89,Z 537.124,A -85,B 0,C 180,E1 -23154.286,E2 -23154.286} C_VEL
LIN {X 0,Y 174.653,Z 531.536,A -85,B 0,C 180,E1 -23157.715,E2 -23157.715} C_VEL
LIN {X 0,Y 179.406,Z 523.847,A -85,B 0,C 180,E1 -23161.27,E2 -23161.27} C_VEL
LIN {X 0,Y 184.337,Z 515.207,A -85,B 0,C 180,E1 -23164.22,E2 -23164.22} C_VEL
LIN {X 0,Y 188.849,Z 506.377,A -85,B 0,C 180,E1 -23166.545,E2 -23166.545} C_VEL
LIN {X 0,Y 193.64,Z 495.532,A -85,B 0,C 180,E1 -23168.762,E2 -23168.762} C_VEL
LIN {X 0,Y 197.714,Z 484.59,A -85,B 0,C 180,E1 -23170.447,E2 -23170.447} C_VEL
LIN {X 0,Y 201.46,Z 472.35,A -85,B 0,C 180,E1 -23171.851,E2 -23171.851} C_VEL
LIN {X 0,Y 204.47,Z 459.435,A -85,B 0,C 180,E1 -23172.923,E2 -23172.923} C_VEL
LIN {X 0,Y 206.585,Z 446.114,A -85,B 0,C 180,E1 -23173.647,E2 -23173.647} C_VEL
LIN {X 0,Y 208.294,Z 424.351,A -85,B 0,C 180,E1 -23174.369,E2 -23174.369} C_VEL
LIN {X 0,Y 209.379,Z 407.488,A -85,B 0,C 180,E1 -23174.9,E2 -23174.9} C_VEL
LIN {X 0,Y 204.509,Z 395.604,A -85,B 0,C 180,E1 -23177.189,E2 -23177.189} C_VEL
LIN {X 0,Y 199.643,Z 385.52,A -85,B 0,C 180,E1 -23179.613,E2 -23179.613} C_VEL
LIN {X 0,Y 195.194,Z 377.259,A -85,B 0,C 180,E1 -23182.021,E2 -23182.021} C_VEL
LIN {X 0,Y 190.758,Z 369.573,A -85,B 0,C 180,E1 -23184.672,E2 -23184.672} C_VEL
LIN {X 0,Y 186.772,Z 363.261,A -85,B 0,C 180,E1 -23187.334,E2 -23187.334} C_VEL
LIN {X 0,Y 183.707,Z 358.652,A -85,B 0,C 180,E1 -23189.622,E2 -23189.622} C_VEL
LIN {X 0,Y 179.35,Z 352.487,A -85,B 0,C 180,E1 -23193.373,E2 -23193.373} C_VEL
LIN {X 0,Y 176.5,Z 349.598,A -85,B 0,C 180,E1 -23196.187,E2 -23196.187} C_VEL
LIN {X 0,Y 175.117,Z 346.949,A -85,B 0,C 180,E1 -23197.932,E2 -23197.932} C_VEL
LIN {X 0,Y 172.452,Z 345.228,A -85,B 0,C 180,E1 -23201.435,E2 -23201.435} C_VEL
LIN {X 0,Y 170.779,Z 342.561,A -85,B 0,C 180,E1 -23204.638,E2 -23204.638} C_VEL
LIN {X 0,Y 170.296,Z 341.09,A -85,B 0,C 180,E1 -23205.969,E2 -23205.969} C_VEL
LIN {X 0,Y 168.469,Z 340.272,A -85,B 0,C 180,E1 -23212.811,E2 -23212.811} C_VEL
LIN {X 0,Y 169.266,Z 340.46,A -85,B 0,C 180,E1 -23220.595,E2 -23220.595} C_VEL
LIN {X 0,Y 170.635,Z 341.279,A -85,B 0,C 180,E1 -23224.208,E2 -23224.208} C_VEL
LIN {X 0,Y 171.844,Z 344.088,A -85,B 0,C 180,E1 -23226.9,E2 -23226.9} C_VEL
LIN {X 0,Y 174.638,Z 346.604,A -85,B 0,C 180,E1 -23230.923,E2 -23230.923} C_VEL
LIN {X 0,Y 175.416,Z 347.209,A -85,B 0,C 180,E1 -23231.849,E2 -23231.849} C_VEL
LIN {X 0,Y 177.142,Z 350.28,A -85,B 0,C 180,E1 -23233.918,E2 -23233.918} C_VEL
LIN {X 0,Y 179.885,Z 352.816,A -85,B 0,C 180,E1 -23236.51,E2 -23236.51} C_VEL
LIN {X 0,Y 182.077,Z 356.116,A -85,B 0,C 180,E1 -23238.462,E2 -23238.462} C_VEL
LIN {X 0,Y 184.124,Z 358.267,A -85,B 0,C 180,E1 -23240.04,E2 -23240.04} C_VEL
LIN {X 0,Y 186.937,Z 361.998,A -85,B 0,C 180,E1 -23242.084,E2 -23242.084} C_VEL
LIN {X 0,Y 191.352,Z 368.113,A -85,B 0,C 180,E1 -23244.949,E2 -23244.949} C_VEL
LIN {X 0,Y 196.388,Z 375.31,A -85,B 0,C 180,E1 -23247.806,E2 -23247.806} C_VEL
LIN {X 0,Y 201.835,Z 384.112,A -85,B 0,C 180,E1 -23250.589,E2 -23250.589} C_VEL
LIN {X 0,Y 206.959,Z 394.338,A -85,B 0,C 180,E1 -23253.023,E2 -23253.023} C_VEL
LIN {X 0,Y 209.818,Z 401.01,A -85,B 0,C 180,E1 -23254.329,E2 -23254.329} C_VEL
LIN {X 0,Y 207.197,Z 436.719,A -85,B 0,C 180,E1 -23255.437,E2 -23255.437} C_VEL
LIN {X 0,Y 205.159,Z 450.484,A -85,B 0,C 180,E1 -23256.175,E2 -23256.175} C_VEL
LIN {X 0,Y 202.483,Z 463.172,A -85,B 0,C 180,E1 -23257.236,E2 -23257.236} C_VEL
LIN {X 0,Y 199.593,Z 473.604,A -85,B 0,C 180,E1 -23258.42,E2 -23258.42} C_VEL
LIN {X 0,Y 195.924,Z 484.535,A -85,B 0,C 180,E1 -23260.056,E2 -23260.056} C_VEL
LIN {X 0,Y 191.683,Z 494.969,A -85,B 0,C 180,E1 -23262.057,E2 -23262.057} C_VEL
LIN {X 0,Y 187.044,Z 504.665,A -85,B 0,C 180,E1 -23264.445,E2 -23264.445} C_VEL
LIN {X 0,Y 182.297,Z 513.328,A -85,B 0,C 180,E1 -23267.243,E2 -23267.243} C_VEL
LIN {X 0,Y 177.331,Z 521.35,A -85,B 0,C 180,E1 -23270.644,E2 -23270.644} C_VEL
LIN {X 0,Y 172.953,Z 527.774,A -85,B 0,C 180,E1 -23274.362,E2 -23274.362} C_VEL
LIN {X 0,Y 168.9,Z 533.083,A -85,B 0,C 180,E1 -23278.657,E2 -23278.657} C_VEL
LIN {X 0,Y 166.088,Z 536.459,A -85,B 0,C 180,E1 -23282.701,E2 -23282.701} C_VEL
LIN {X 0,Y 163.768,Z 538.708,A -85,B 0,C 180,E1 -23287.278,E2 -23287.278} C_VEL
LIN {X 0,Y 162.295,Z 539.576,A -85,B 0,C 180,E1 -23292.353,E2 -23292.353} C_VEL
LIN {X 0,Y 161.845,Z 539.381,A -85,B 0,C 180,E1 -23294.896,E2 -23294.896} C_VEL
LIN {X 0,Y 161.576,Z 538.768,A -85,B 0,C 180,E1 -23297.437,E2 -23297.437} C_VEL
LIN {X 0,Y 161.532,Z 537.761,A -85,B 0,C 180,E1 -23299.976,E2 -23299.976} C_VEL
LIN {X 0,Y 161.691,Z 536.354,A -85,B 0,C 180,E1 -23302.506,E2 -23302.506} C_VEL
LIN {X 0,Y 162.141,Z 534.044,A -85,B 0,C 180,E1 -23305.525,E2 -23305.525} C_VEL
LIN {X 0,Y 162.955,Z 529.43,A -85,B 0,C 180,E1 -23309.998,E2 -23309.998} C_VEL
LIN {X 0,Y 164.456,Z 523.315,A -85,B 0,C 180,E1 -23314.287,E2 -23314.287} C_VEL
LIN {X 0,Y 166.34,Z 516.638,A -85,B 0,C 180,E1 -23317.891,E2 -23317.891} C_VEL
LIN {X 0,Y 168.738,Z 508.36,A -85,B 0,C 180,E1 -23321.409,E2 -23321.409} C_VEL
LIN {X 0,Y 171.11,Z 499.861,A -85,B 0,C 180,E1 -23324.265,E2 -23324.265} C_VEL
LIN {X 0,Y 173.776,Z 490.498,A -85,B 0,C 180,E1 -23326.746,E2 -23326.746} C_VEL
LIN {X 0,Y 176.344,Z 480.314,A -85,B 0,C 180,E1 -23328.892,E2 -23328.892} C_VEL
LIN {X 0,Y 178.583,Z 469.247,A -85,B 0,C 180,E1 -23330.742,E2 -23330.742} C_VEL
LIN {X 0,Y 180.567,Z 456.965,A -85,B 0,C 180,E1 -23332.3,E2 -23332.3} C_VEL
LIN {X 0,Y 182.165,Z 443.442,A -85,B 0,C 180,E1 -23333.481,E2 -23333.481} C_VEL
LIN {X 0,Y 183.212,Z 429.907,A -85,B 0,C 180,E1 -23334.2,E2 -23334.2} C_VEL
LIN {X 0,Y 185.766,Z 377.532,A -85,B 0,C 180,E1 -23336.076,E2 -23336.076} C_VEL
LIN {X 0,Y 181.247,Z 365.61,A -85,B 0,C 180,E1 -23337.552,E2 -23337.552} C_VEL
LIN {X 0,Y 174.435,Z 352.489,A -85,B 0,C 180,E1 -23339.729,E2 -23339.729} C_VEL
LIN {X 0,Y 168.701,Z 342.834,A -85,B 0,C 180,E1 -23341.672,E2 -23341.672} C_VEL
LIN {X 0,Y 166.357,Z 339.111,A -85,B 0,C 180,E1 -23342.508,E2 -23342.508} C_VEL
LIN {X 0,Y 164.816,Z 336.878,A -85,B 0,C 180,E1 -23343.065,E2 -23343.065} C_VEL
LIN {X 0,Y 164.326,Z 335.011,A -85,B 0,C 180,E1 -23343.352,E2 -23343.352} C_VEL
LIN {X 0,Y 164.277,Z 335.018,A -85,B 0,C 180,E1 -23346.791,E2 -23346.791} C_VEL
LIN {X 0,Y 164.283,Z 335.011,A -85,B 0,C 180,E1 -23349.916,E2 -23349.916} C_VEL
LIN {X 0,Y 164.277,Z 335.022,A -85,B 0,C 180,E1 -23353.34,E2 -23353.34} C_VEL
LIN {X 0,Y 164.256,Z 335.006,A -85,B 0,C 180,E1 -23356.796,E2 -23356.796} C_VEL
LIN {X 0,Y 164.285,Z 335.017,A -85,B 0,C 180,E1 -23360.353,E2 -23360.353} C_VEL
LIN {X 0,Y 164.321,Z 334.993,A -85,B 0,C 180,E1 -23364.35,E2 -23364.35} C_VEL
LIN {X 0,Y 164.365,Z 335.009,A -85,B 0,C 180,E1 -23369.129,E2 -23369.129} C_VEL
LIN {X 0,Y 164.352,Z 334.984,A -85,B 0,C 180,E1 -23374.683,E2 -23374.683} C_VEL
LIN {X 0,Y 164.411,Z 335.004,A -85,B 0,C 180,E1 -23380.116,E2 -23380.116} C_VEL
LIN {X 0,Y 164.459,Z 334.969,A -85,B 0,C 180,E1 -23385.143,E2 -23385.143} C_VEL
LIN {X 0,Y 164.756,Z 334.962,A -85,B 0,C 180,E1 -23390.175,E2 -23390.175} C_VEL
LIN {X 0,Y 164.81,Z 334.944,A -85,B 0,C 180,E1 -23392.65,E2 -23392.65} C_VEL
LIN {X 0,Y 165.267,Z 334.897,A -85,B 0,C 180,E1 -23400,E2 -23400} C_VEL
LIN {X 0,Y 164.815,Z 334.934,A -85,B 0,C 180,E1 -23407.349,E2 -23407.349} C_VEL
LIN {X 0,Y 164.695,Z 334.969,A -85,B 0,C 180,E1 -23411.059,E2 -23411.059} C_VEL
LIN {X 0,Y 164.445,Z 334.984,A -85,B 0,C 180,E1 -23417.407,E2 -23417.407} C_VEL
LIN {X 0,Y 164.443,Z 335.001,A -85,B 0,C 180,E1 -23419.993,E2 -23419.993} C_VEL
LIN {X 0,Y 164.379,Z 335.008,A -85,B 0,C 180,E1 -23426.128,E2 -23426.128} C_VEL
LIN {X 0,Y 164.368,Z 335.01,A -85,B 0,C 180,E1 -23431.228,E2 -23431.228} C_VEL
LIN {X 0,Y 164.274,Z 335.017,A -85,B 0,C 180,E1 -23436.794,E2 -23436.794} C_VEL
LIN {X 0,Y 164.281,Z 335.018,A -85,B 0,C 180,E1 -23439.919,E2 -23439.919} C_VEL
LIN {X 0,Y 164.314,Z 335.186,A -85,B 0,C 180,E1 -23445.104,E2 -23445.104} C_VEL
LIN {X 0,Y 164.424,Z 335.707,A -85,B 0,C 180,E1 -23445.391,E2 -23445.391} C_VEL
LIN {X 0,Y 165.725,Z 338.44,A -85,B 0,C 180,E1 -23445.912,E2 -23445.912} C_VEL
LIN {X 0,Y 167.557,Z 341.539,A -85,B 0,C 180,E1 -23446.585,E2 -23446.585} C_VEL
LIN {X 0,Y 173.367,Z 352.638,A -85,B 0,C 180,E1 -23448.653,E2 -23448.653} C_VEL
LIN {X 0,Y 179.196,Z 366.306,A -85,B 0,C 180,E1 -23450.672,E2 -23450.672} C_VEL
LIN {X 0,Y 183.599,Z 378.397,A -85,B 0,C 180,E1 -23452.166,E2 -23452.166} C_VEL
LIN {X 0,Y 185.09,Z 396.122,A -85,B 0,C 180,E1 -23453.265,E2 -23453.265} C_VEL
LIN {X 0,Y 182.667,Z 445.135,A -85,B 0,C 180,E1 -23455.091,E2 -23455.091} C_VEL
LIN {X 0,Y 181.162,Z 458.982,A -85,B 0,C 180,E1 -23456.024,E2 -23456.024} C_VEL
LIN {X 0,Y 179.111,Z 471.893,A -85,B 0,C 180,E1 -23457.351,E2 -23457.351} C_VEL
LIN {X 0,Y 176.581,Z 484.492,A -85,B 0,C 180,E1 -23459.176,E2 -23459.176} C_VEL
LIN {X 0,Y 173.903,Z 495.717,A -85,B 0,C 180,E1 -23461.323,E2 -23461.323} C_VEL
LIN {X 0,Y 171.649,Z 503.736,A -85,B 0,C 180,E1 -23463.244,E2 -23463.244} C_VEL
LIN {X 0,Y 169.97,Z 508.193,A -85,B 0,C 180,E1 -23464.421,E2 -23464.421} C_VEL
LIN {X 0,Y 165.38,Z 515.016,A -85,B 0,C 180,E1 -23466.33,E2 -23466.33} C_VEL
LIN {X 0,Y 160.743,Z 521.241,A -85,B 0,C 180,E1 -23468.527,E2 -23468.527} C_VEL
LIN {X 0,Y 159.046,Z 524.763,A -85,B 0,C 180,E1 -23470.126,E2 -23470.126} C_VEL
LIN {X 0,Y 156.799,Z 532.406,A -85,B 0,C 180,E1 -23474.402,E2 -23474.402} C_VEL
LIN {X 0,Y 155.634,Z 537.727,A -85,B 0,C 180,E1 -23478.277,E2 -23478.277} C_VEL
LIN {X 0,Y 154.963,Z 541.844,A -85,B 0,C 180,E1 -23482.182,E2 -23482.182} C_VEL
LIN {X 0,Y 154.754,Z 543.984,A -85,B 0,C 180,E1 -23484.791,E2 -23484.791} C_VEL
LIN {X 0,Y 154.738,Z 545.841,A -85,B 0,C 180,E1 -23487.721,E2 -23487.721} C_VEL
LIN {X 0,Y 154.852,Z 546.928,A -85,B 0,C 180,E1 -23490.002,E2 -23490.002} C_VEL
LIN {X 0,Y 154.736,Z 547.782,A -85,B 0,C 180,E1 -23492.605,E2 -23492.605} C_VEL
LIN {X 0,Y 154.757,Z 548.206,A -85,B 0,C 180,E1 -23495.213,E2 -23495.213} C_VEL
LIN {X 0,Y 155.453,Z 547.881,A -85,B 0,C 180,E1 -23500.42,E2 -23500.42} C_VEL
LIN {X 0,Y 156.207,Z 547.152,A -85,B 0,C 180,E1 -23503.002,E2 -23503.002} C_VEL
LIN {X 0,Y 157.216,Z 546.017,A -85,B 0,C 180,E1 -23505.56,E2 -23505.56} C_VEL
LIN {X 0,Y 158.506,Z 544.453,A -85,B 0,C 180,E1 -23508.083,E2 -23508.083} C_VEL
LIN {X 0,Y 161.188,Z 541.34,A -85,B 0,C 180,E1 -23511.755,E2 -23511.755} C_VEL
LIN {X 0,Y 164.443,Z 537.192,A -85,B 0,C 180,E1 -23515.303,E2 -23515.303} C_VEL
LIN {X 0,Y 168.839,Z 531.019,A -85,B 0,C 180,E1 -23519.199,E2 -23519.199} C_VEL
LIN {X 0,Y 173.368,Z 524.066,A -85,B 0,C 180,E1 -23522.49,E2 -23522.49} C_VEL
LIN {X 0,Y 178.535,Z 515.557,A -85,B 0,C 180,E1 -23525.497,E2 -23525.497} C_VEL
LIN {X 0,Y 183.22,Z 506.839,A -85,B 0,C 180,E1 -23527.861,E2 -23527.861} C_VEL
LIN {X 0,Y 188.175,Z 496.135,A -85,B 0,C 180,E1 -23530.112,E2 -23530.112} C_VEL
LIN {X 0,Y 192.404,Z 485.457,A -85,B 0,C 180,E1 -23531.808,E2 -23531.808} C_VEL
LIN {X 0,Y 196.262,Z 473.497,A -85,B 0,C 180,E1 -23533.226,E2 -23533.226} C_VEL
LIN {X 0,Y 199.384,Z 461.056,A -85,B 0,C 180,E1 -23534.297,E2 -23534.297} C_VEL
LIN {X 0,Y 201.558,Z 448.917,A -85,B 0,C 180,E1 -23535.026,E2 -23535.026} C_VEL
LIN {X 0,Y 202.949,Z 434.849,A -85,B 0,C 180,E1 -23535.56,E2 -23535.56} C_VEL
LIN {X 0,Y 204.65,Z 409.822,A -85,B 0,C 180,E1 -23536.349,E2 -23536.349} C_VEL
LIN {X 0,Y 200.09,Z 398.645,A -85,B 0,C 180,E1 -23538.648,E2 -23538.648} C_VEL
LIN {X 0,Y 195.326,Z 388.547,A -85,B 0,C 180,E1 -23541.223,E2 -23541.223} C_VEL
LIN {X 0,Y 190.015,Z 378.735,A -85,B 0,C 180,E1 -23544.381,E2 -23544.381} C_VEL
LIN {X 0,Y 185.118,Z 370.29,A -85,B 0,C 180,E1 -23547.732,E2 -23547.732} C_VEL
LIN {X 0,Y 181.445,Z 364.691,A -85,B 0,C 180,E1 -23550.593,E2 -23550.593} C_VEL
LIN {X 0,Y 177.661,Z 359.053,A -85,B 0,C 180,E1 -23554.048,E2 -23554.048} C_VEL
LIN {X 0,Y 174.951,Z 356.219,A -85,B 0,C 180,E1 -23556.858,E2 -23556.858} C_VEL
LIN {X 0,Y 173.624,Z 353.786,A -85,B 0,C 180,E1 -23558.594,E2 -23558.594} C_VEL
LIN {X 0,Y 170.979,Z 351.759,A -85,B 0,C 180,E1 -23562.354,E2 -23562.354} C_VEL
LIN {X 0,Y 169.539,Z 349.112,A -85,B 0,C 180,E1 -23565.445,E2 -23565.445} C_VEL
LIN {X 0,Y 169.126,Z 348.068,A -85,B 0,C 180,E1 -23566.636,E2 -23566.636} C_VEL
LIN {X 0,Y 167.601,Z 347.319,A -85,B 0,C 180,E1 -23572.774,E2 -23572.774} C_VEL
LIN {X 0,Y 168.392,Z 347.505,A -85,B 0,C 180,E1 -23580.598,E2 -23580.598} C_VEL
LIN {X 0,Y 169.515,Z 348.283,A -85,B 0,C 180,E1 -23583.715,E2 -23583.715} C_VEL
LIN {X 0,Y 171.139,Z 351.589,A -85,B 0,C 180,E1 -23587.276,E2 -23587.276} C_VEL
LIN {X 0,Y 173.891,Z 353.923,A -85,B 0,C 180,E1 -23591.152,E2 -23591.152} C_VEL
LIN {X 0,Y 175.93,Z 357.323,A -85,B 0,C 180,E1 -23593.648,E2 -23593.648} C_VEL
LIN {X 0,Y 178.132,Z 359.455,A -85,B 0,C 180,E1 -23595.812,E2 -23595.812} C_VEL
LIN {X 0,Y 180.669,Z 363.098,A -85,B 0,C 180,E1 -23598.132,E2 -23598.132} C_VEL
LIN {X 0,Y 182.072,Z 364.647,A -85,B 0,C 180,E1 -23599.259,E2 -23599.259} C_VEL
LIN {X 0,Y 185.934,Z 370.036,A -85,B 0,C 180,E1 -23602.155,E2 -23602.155} C_VEL
LIN {X 0,Y 189.281,Z 374.829,A -85,B 0,C 180,E1 -23604.38,E2 -23604.38} C_VEL
LIN {X 0,Y 194.012,Z 381.86,A -85,B 0,C 180,E1 -23607.178,E2 -23607.178} C_VEL
LIN {X 0,Y 198.536,Z 389.393,A -85,B 0,C 180,E1 -23609.604,E2 -23609.604} C_VEL
LIN {X 0,Y 203.417,Z 399.554,A -85,B 0,C 180,E1 -23612.069,E2 -23612.069} C_VEL
LIN {X 0,Y 205.092,Z 403.318,A -85,B 0,C 180,E1 -23612.872,E2 -23612.872} C_VEL
LIN {X 0,Y 202.576,Z 436.827,A -85,B 0,C 180,E1 -23613.934,E2 -23613.934} C_VEL
LIN {X 0,Y 200.547,Z 450.221,A -85,B 0,C 180,E1 -23614.648,E2 -23614.648} C_VEL
LIN {X 0,Y 197.857,Z 462.576,A -85,B 0,C 180,E1 -23615.654,E2 -23615.654} C_VEL
LIN {X 0,Y 194.603,Z 474.024,A -85,B 0,C 180,E1 -23616.96,E2 -23616.96} C_VEL
LIN {X 0,Y 190.841,Z 484.783,A -85,B 0,C 180,E1 -23618.588,E2 -23618.588} C_VEL
LIN {X 0,Y 186.367,Z 495.342,A -85,B 0,C 180,E1 -23620.638,E2 -23620.638} C_VEL
LIN {X 0,Y 182.006,Z 504.091,A -85,B 0,C 180,E1 -23622.804,E2 -23622.804} C_VEL
LIN {X 0,Y 177.015,Z 512.881,A -85,B 0,C 180,E1 -23625.616,E2 -23625.616} C_VEL
LIN {X 0,Y 171.728,Z 521.052,A -85,B 0,C 180,E1 -23629.094,E2 -23629.094} C_VEL
LIN {X 0,Y 167.544,Z 526.969,A -85,B 0,C 180,E1 -23632.471,E2 -23632.471} C_VEL
LIN {X 0,Y 163.755,Z 531.731,A -85,B 0,C 180,E1 -23636.085,E2 -23636.085} C_VEL
LIN {X 0,Y 161.673,Z 534.183,A -85,B 0,C 180,E1 -23638.556,E2 -23638.556} C_VEL
LIN {X 0,Y 159.314,Z 536.753,A -85,B 0,C 180,E1 -23641.92,E2 -23641.92} C_VEL
LIN {X 0,Y 157.031,Z 538.822,A -85,B 0,C 180,E1 -23646.245,E2 -23646.245} C_VEL
LIN {X 0,Y 155.344,Z 539.762,A -85,B 0,C 180,E1 -23651.535,E2 -23651.535} C_VEL
LIN {X 0,Y 154.836,Z 539.633,A -85,B 0,C 180,E1 -23654.195,E2 -23654.195} C_VEL
LIN {X 0,Y 154.524,Z 539.059,A -85,B 0,C 180,E1 -23656.854,E2 -23656.854} C_VEL
LIN {X 0,Y 154.431,Z 538.088,A -85,B 0,C 180,E1 -23659.51,E2 -23659.51} C_VEL
LIN {X 0,Y 154.557,Z 536.72,A -85,B 0,C 180,E1 -23662.158,E2 -23662.158} C_VEL
LIN {X 0,Y 155.058,Z 534.181,A -85,B 0,C 180,E1 -23665.682,E2 -23665.682} C_VEL
LIN {X 0,Y 155.853,Z 529.942,A -85,B 0,C 180,E1 -23669.998,E2 -23669.998} C_VEL
LIN {X 0,Y 157.129,Z 524.916,A -85,B 0,C 180,E1 -23673.845,E2 -23673.845} C_VEL
LIN {X 0,Y 158.905,Z 518.608,A -85,B 0,C 180,E1 -23677.623,E2 -23677.623} C_VEL
LIN {X 0,Y 161.362,Z 510.694,A -85,B 0,C 180,E1 -23681.301,E2 -23681.301} C_VEL
LIN {X 0,Y 163.701,Z 502.652,A -85,B 0,C 180,E1 -23684.29,E2 -23684.29} C_VEL
LIN {X 0,Y 166.61,Z 492.813,A -85,B 0,C 180,E1 -23687.172,E2 -23687.172} C_VEL
LIN {X 0,Y 169.36,Z 483.119,A -85,B 0,C 180,E1 -23689.387,E2 -23689.387} C_VEL
LIN {X 0,Y 171.667,Z 472.731,A -85,B 0,C 180,E1 -23691.303,E2 -23691.303} C_VEL
LIN {X 0,Y 173.906,Z 460.271,A -85,B 0,C 180,E1 -23693.046,E2 -23693.046} C_VEL
LIN {X 0,Y 175.686,Z 447.141,A -85,B 0,C 180,E1 -23694.362,E2 -23694.362} C_VEL
LIN {X 0,Y 176.885,Z 433.851,A -85,B 0,C 180,E1 -23695.204,E2 -23695.204} C_VEL
LIN {X 0,Y 179.765,Z 380.258,A -85,B 0,C 180,E1 -23697.175,E2 -23697.175} C_VEL
LIN {X 0,Y 179.217,Z 377.835,A -85,B 0,C 180,E1 -23697.407,E2 -23697.407} C_VEL
LIN {X 0,Y 175.71,Z 368.677,A -85,B 0,C 180,E1 -23698.626,E2 -23698.626} C_VEL
LIN {X 0,Y 168.646,Z 355.047,A -85,B 0,C 180,E1 -23701.038,E2 -23701.038} C_VEL
LIN {X 0,Y 162.117,Z 344.229,A -85,B 0,C 180,E1 -23703.433,E2 -23703.433} C_VEL
LIN {X 0,Y 160.044,Z 340.927,A -85,B 0,C 180,E1 -23704.245,E2 -23704.245} C_VEL
LIN {X 0,Y 157.856,Z 337.933,A -85,B 0,C 180,E1 -23705.108,E2 -23705.108} C_VEL
LIN {X 0,Y 157.271,Z 335.891,A -85,B 0,C 180,E1 -23705.462,E2 -23705.462} C_VEL
LIN {X 0,Y 157.191,Z 335.892,A -85,B 0,C 180,E1 -23710.529,E2 -23710.529} C_VEL
LIN {X 0,Y 157.175,Z 335.894,A -85,B 0,C 180,E1 -23715.675,E2 -23715.675} C_VEL
LIN {X 0,Y 157.194,Z 335.901,A -85,B 0,C 180,E1 -23721.249,E2 -23721.249} C_VEL
LIN {X 0,Y 157.27,Z 335.869,A -85,B 0,C 180,E1 -23724.483,E2 -23724.483} C_VEL
LIN {X 0,Y 157.278,Z 335.889,A -85,B 0,C 180,E1 -23728.1,E2 -23728.1} C_VEL
LIN {X 0,Y 157.261,Z 335.867,A -85,B 0,C 180,E1 -23733.454,E2 -23733.454} C_VEL
LIN {X 0,Y 157.353,Z 335.885,A -85,B 0,C 180,E1 -23739.701,E2 -23739.701} C_VEL
LIN {X 0,Y 157.394,Z 335.847,A -85,B 0,C 180,E1 -23744.459,E2 -23744.459} C_VEL
LIN {X 0,Y 157.678,Z 335.843,A -85,B 0,C 180,E1 -23749.729,E2 -23749.729} C_VEL
LIN {X 0,Y 157.749,Z 335.825,A -85,B 0,C 180,E1 -23752.319,E2 -23752.319} C_VEL
LIN {X 0,Y 158.229,Z 335.773,A -85,B 0,C 180,E1 -23760,E2 -23760} C_VEL
LIN {X 0,Y 157.753,Z 335.816,A -85,B 0,C 180,E1 -23767.68,E2 -23767.68} C_VEL
LIN {X 0,Y 157.626,Z 335.85,A -85,B 0,C 180,E1 -23771.228,E2 -23771.228} C_VEL
LIN {X 0,Y 157.414,Z 335.85,A -85,B 0,C 180,E1 -23775.538,E2 -23775.538} C_VEL
LIN {X 0,Y 157.351,Z 335.884,A -85,B 0,C 180,E1 -23780.935,E2 -23780.935} C_VEL
LIN {X 0,Y 157.304,Z 335.889,A -85,B 0,C 180,E1 -23786.681,E2 -23786.681} C_VEL
LIN {X 0,Y 157.269,Z 335.888,A -85,B 0,C 180,E1 -23792.429,E2 -23792.429} C_VEL
LIN {X 0,Y 157.253,Z 335.892,A -85,B 0,C 180,E1 -23796.446,E2 -23796.446} C_VEL
LIN {X 0,Y 157.185,Z 335.887,A -85,B 0,C 180,E1 -23802.119,E2 -23802.119} C_VEL
LIN {X 0,Y 157.215,Z 335.886,A -85,B 0,C 180,E1 -23803.18,E2 -23803.18} C_VEL
LIN {X 0,Y 158.352,Z 338.897,A -85,B 0,C 180,E1 -23803.744,E2 -23803.744} C_VEL
LIN {X 0,Y 160.119,Z 341.126,A -85,B 0,C 180,E1 -23804.424,E2 -23804.424} C_VEL
LIN {X 0,Y 163.147,Z 346.499,A -85,B 0,C 180,E1 -23805.628,E2 -23805.628} C_VEL
LIN {X 0,Y 168.686,Z 357.37,A -85,B 0,C 180,E1 -23807.726,E2 -23807.726} C_VEL
LIN {X 0,Y 174.023,Z 370.131,A -85,B 0,C 180,E1 -23809.688,E2 -23809.688} C_VEL
LIN {X 0,Y 177.79,Z 380.637,A -85,B 0,C 180,E1 -23811.053,E2 -23811.053} C_VEL
LIN {X 0,Y 179.079,Z 395.816,A -85,B 0,C 180,E1 -23812.05,E2 -23812.05} C_VEL
LIN {X 0,Y 176.6,Z 444.161,A -85,B 0,C 180,E1 -23813.882,E2 -23813.882} C_VEL
LIN {X 0,Y 175.198,Z 457.522,A -85,B 0,C 180,E1 -23814.787,E2 -23814.787} C_VEL
LIN {X 0,Y 173.159,Z 470.301,A -85,B 0,C 180,E1 -23816.08,E2 -23816.08} C_VEL
LIN {X 0,Y 170.88,Z 481.644,A -85,B 0,C 180,E1 -23817.681,E2 -23817.681} C_VEL
LIN {X 0,Y 167.912,Z 493.337,A -85,B 0,C 180,E1 -23819.852,E2 -23819.852} C_VEL
LIN {X 0,Y 165.002,Z 503.868,A -85,B 0,C 180,E1 -23822.408,E2 -23822.408} C_VEL
LIN {X 0,Y 162.51,Z 512.983,A -85,B 0,C 180,E1 -23825.254,E2 -23825.254} C_VEL
LIN {X 0,Y 160.379,Z 520.42,A -85,B 0,C 180,E1 -23828.133,E2 -23828.133} C_VEL
LIN {X 0,Y 159.046,Z 524.763,A -85,B 0,C 180,E1 -23830.126,E2 -23830.126} C_VEL
LIN {X 0,Y 157.456,Z 528.105,A -85,B 0,C 180,E1 -23831.808,E2 -23831.808} C_VEL
LIN {X 0,Y 153.282,Z 532.984,A -85,B 0,C 180,E1 -23834.598,E2 -23834.598} C_VEL
LIN {X 0,Y 149.37,Z 537.177,A -85,B 0,C 180,E1 -23837.663,E2 -23837.663} C_VEL
LIN {X 0,Y 148.235,Z 539.434,A -85,B 0,C 180,E1 -23839.717,E2 -23839.717} C_VEL
LIN {X 0,Y 147.688,Z 543.636,A -85,B 0,C 180,E1 -23844.541,E2 -23844.541} C_VEL
LIN {X 0,Y 147.658,Z 545.848,A -85,B 0,C 180,E1 -23848.226,E2 -23848.226} C_VEL
LIN {X 0,Y 147.765,Z 546.637,A -85,B 0,C 180,E1 -23850.002,E2 -23850.002} C_VEL
LIN {X 0,Y 147.643,Z 547.518,A -85,B 0,C 180,E1 -23852.73,E2 -23852.73} C_VEL
LIN {X 0,Y 147.689,Z 547.993,A -85,B 0,C 180,E1 -23855.463,E2 -23855.463} C_VEL
LIN {X 0,Y 148.443,Z 547.721,A -85,B 0,C 180,E1 -23860.918,E2 -23860.918} C_VEL
LIN {X 0,Y 150.348,Z 545.931,A -85,B 0,C 180,E1 -23866.29,E2 -23866.29} C_VEL
LIN {X 0,Y 151.756,Z 544.404,A -85,B 0,C 180,E1 -23868.918,E2 -23868.918} C_VEL
LIN {X 0,Y 154.607,Z 541.351,A -85,B 0,C 180,E1 -23872.732,E2 -23872.732} C_VEL
LIN {X 0,Y 158.054,Z 537.267,A -85,B 0,C 180,E1 -23876.403,E2 -23876.403} C_VEL
LIN {X 0,Y 162.534,Z 531.346,A -85,B 0,C 180,E1 -23880.318,E2 -23880.318} C_VEL
LIN {X 0,Y 167.425,Z 524.285,A -85,B 0,C 180,E1 -23883.795,E2 -23883.795} C_VEL
LIN {X 0,Y 172.826,Z 515.909,A -85,B 0,C 180,E1 -23886.858,E2 -23886.858} C_VEL
LIN {X 0,Y 177.68,Z 507.304,A -85,B 0,C 180,E1 -23889.264,E2 -23889.264} C_VEL
LIN {X 0,Y 182.832,Z 496.732,A -85,B 0,C 180,E1 -23891.537,E2 -23891.537} C_VEL
LIN {X 0,Y 187.21,Z 486.247,A -85,B 0,C 180,E1 -23893.246,E2 -23893.246} C_VEL
LIN {X 0,Y 191.206,Z 474.638,A -85,B 0,C 180,E1 -23894.667,E2 -23894.667} C_VEL
LIN {X 0,Y 194.694,Z 461.326,A -85,B 0,C 180,E1 -23895.845,E2 -23895.845} C_VEL
LIN {X 0,Y 197.087,Z 448.551,A -85,B 0,C 180,E1 -23896.61,E2 -23896.61} C_VEL
LIN {X 0,Y 198.546,Z 434.038,A -85,B 0,C 180,E1 -23897.157,E2 -23897.157} C_VEL
LIN {X 0,Y 200.088,Z 412.335,A -85,B 0,C 180,E1 -23897.845,E2 -23897.845} C_VEL
LIN {X 0,Y 195.707,Z 401.521,A -85,B 0,C 180,E1 -23900.23,E2 -23900.23} C_VEL
LIN {X 0,Y 191.505,Z 392.524,A -85,B 0,C 180,E1 -23902.681,E2 -23902.681} C_VEL
LIN {X 0,Y 186.973,Z 383.895,A -85,B 0,C 180,E1 -23905.586,E2 -23905.586} C_VEL
LIN {X 0,Y 182.62,Z 376.065,A -85,B 0,C 180,E1 -23908.78,E2 -23908.78} C_VEL
LIN {X 0,Y 179.289,Z 370.79,A -85,B 0,C 180,E1 -23911.542,E2 -23911.542} C_VEL
LIN {X 0,Y 175.906,Z 365.593,A -85,B 0,C 180,E1 -23914.816,E2 -23914.816} C_VEL
LIN {X 0,Y 173.39,Z 362.762,A -85,B 0,C 180,E1 -23917.588,E2 -23917.588} C_VEL
LIN {X 0,Y 172.315,Z 360.689,A -85,B 0,C 180,E1 -23919.071,E2 -23919.071} C_VEL
LIN {X 0,Y 169.525,Z 358.242,A -85,B 0,C 180,E1 -23923.363,E2 -23923.363} C_VEL
LIN {X 0,Y 168.311,Z 355.619,A -85,B 0,C 180,E1 -23926.339,E2 -23926.339} C_VEL
LIN {X 0,Y 167.983,Z 355.032,A -85,B 0,C 180,E1 -23927.312,E2 -23927.312} C_VEL
LIN {X 0,Y 166.733,Z 354.37,A -85,B 0,C 180,E1 -23932.736,E2 -23932.736} C_VEL
LIN {X 0,Y 167.356,Z 354.434,A -85,B 0,C 180,E1 -23940,E2 -23940} C_VEL
LIN {X 0,Y 168.425,Z 355.227,A -85,B 0,C 180,E1 -23943.234,E2 -23943.234} C_VEL
LIN {X 0,Y 170.029,Z 358.509,A -85,B 0,C 180,E1 -23946.922,E2 -23946.922} C_VEL
LIN {X 0,Y 172.458,Z 360.749,A -85,B 0,C 180,E1 -23950.53,E2 -23950.53} C_VEL
LIN {X 0,Y 174.468,Z 364.066,A -85,B 0,C 180,E1 -23953.097,E2 -23953.097} C_VEL
LIN {X 0,Y 176.396,Z 365.995,A -85,B 0,C 180,E1 -23955.084,E2 -23955.084} C_VEL
LIN {X 0,Y 178.961,Z 369.733,A -85,B 0,C 180,E1 -23957.535,E2 -23957.535} C_VEL
LIN {X 0,Y 180.278,Z 371.38,A -85,B 0,C 180,E1 -23958.653,E2 -23958.653} C_VEL
LIN {X 0,Y 183.63,Z 376.155,A -85,B 0,C 180,E1 -23961.285,E2 -23961.285} C_VEL
LIN {X 0,Y 186.8,Z 380.842,A -85,B 0,C 180,E1 -23963.508,E2 -23963.508} C_VEL
LIN {X 0,Y 191.719,Z 388.395,A -85,B 0,C 180,E1 -23966.561,E2 -23966.561} C_VEL
LIN {X 0,Y 195.541,Z 395.145,A -85,B 0,C 180,E1 -23968.72,E2 -23968.72} C_VEL
LIN {X 0,Y 200.162,Z 405.19,A -85,B 0,C 180,E1 -23971.192,E2 -23971.192} C_VEL
LIN {X 0,Y 200.546,Z 406.148,A -85,B 0,C 180,E1 -23971.393,E2 -23971.393} C_VEL
LIN {X 0,Y 197.992,Z 437.764,A -85,B 0,C 180,E1 -23972.396,E2 -23972.396} C_VEL
LIN {X 0,Y 195.893,Z 450.941,A -85,B 0,C 180,E1 -23973.114,E2 -23973.114} C_VEL
LIN {X 0,Y 193.125,Z 463.082,A -85,B 0,C 180,E1 -23974.115,E2 -23974.115} C_VEL
LIN {X 0,Y 189.746,Z 474.445,A -85,B 0,C 180,E1 -23975.425,E2 -23975.425} C_VEL
LIN {X 0,Y 185.938,Z 484.895,A -85,B 0,C 180,E1 -23977.014,E2 -23977.014} C_VEL
LIN {X 0,Y 181.184,Z 495.664,A -85,B 0,C 180,E1 -23979.122,E2 -23979.122} C_VEL
LIN {X 0,Y 176.14,Z 505.294,A -85,B 0,C 180,E1 -23981.57,E2 -23981.57} C_VEL
LIN {X 0,Y 170.805,Z 514.108,A -85,B 0,C 180,E1 -23984.536,E2 -23984.536} C_VEL
LIN {X 0,Y 165.449,Z 521.897,A -85,B 0,C 180,E1 -23988.006,E2 -23988.006} C_VEL
LIN {X 0,Y 161.568,Z 527.033,A -85,B 0,C 180,E1 -23991.055,E2 -23991.055} C_VEL
LIN {X 0,Y 157.718,Z 531.62,A -85,B 0,C 180,E1 -23994.598,E2 -23994.598} C_VEL
LIN {X 0,Y 154.432,Z 535.227,A -85,B 0,C 180,E1 -23998.441,E2 -23998.441} C_VEL
LIN {X 0,Y 151.771,Z 537.773,A -85,B 0,C 180,E1 -24002.413,E2 -24002.413} C_VEL
LIN {X 0,Y 150.349,Z 538.935,A -85,B 0,C 180,E1 -24005.119,E2 -24005.119} C_VEL
LIN {X 0,Y 148.421,Z 539.948,A -85,B 0,C 180,E1 -24010.641,E2 -24010.641} C_VEL
LIN {X 0,Y 147.856,Z 539.862,A -85,B 0,C 180,E1 -24013.427,E2 -24013.427} C_VEL
LIN {X 0,Y 147.492,Z 539.351,A -85,B 0,C 180,E1 -24016.215,E2 -24016.215} C_VEL
LIN {X 0,Y 147.353,Z 538.414,A -85,B 0,C 180,E1 -24019,E2 -24019} C_VEL
LIN {X 0,Y 147.425,Z 537.083,A -85,B 0,C 180,E1 -24021.776,E2 -24021.776} C_VEL
LIN {X 0,Y 147.985,Z 534.347,A -85,B 0,C 180,E1 -24025.815,E2 -24025.815} C_VEL
LIN {X 0,Y 148.753,Z 530.453,A -85,B 0,C 180,E1 -24029.998,E2 -24029.998} C_VEL
LIN {X 0,Y 150.046,Z 525.512,A -85,B 0,C 180,E1 -24034.027,E2 -24034.027} C_VEL
LIN {X 0,Y 151.878,Z 519.304,A -85,B 0,C 180,E1 -24037.978,E2 -24037.978} C_VEL
LIN {X 0,Y 154.418,Z 511.545,A -85,B 0,C 180,E1 -24041.816,E2 -24041.816} C_VEL
LIN {X 0,Y 157.421,Z 501.847,A -85,B 0,C 180,E1 -24045.535,E2 -24045.535} C_VEL
LIN {X 0,Y 160.527,Z 491.786,A -85,B 0,C 180,E1 -24048.504,E2 -24048.504} C_VEL
LIN {X 0,Y 163.38,Z 481.781,A -85,B 0,C 180,E1 -24050.784,E2 -24050.784} C_VEL
LIN {X 0,Y 166.194,Z 469.203,A -85,B 0,C 180,E1 -24053.025,E2 -24053.025} C_VEL
LIN {X 0,Y 168.371,Z 456.731,A -85,B 0,C 180,E1 -24054.669,E2 -24054.669} C_VEL
LIN {X 0,Y 170.059,Z 443.403,A -85,B 0,C 180,E1 -24055.88,E2 -24055.88} C_VEL
LIN {X 0,Y 171.142,Z 430.304,A -85,B 0,C 180,E1 -24056.605,E2 -24056.605} C_VEL
LIN {X 0,Y 173.753,Z 380.965,A -85,B 0,C 180,E1 -24058.466,E2 -24058.466} C_VEL
LIN {X 0,Y 170.518,Z 372.427,A -85,B 0,C 180,E1 -24059.662,E2 -24059.662} C_VEL
LIN {X 0,Y 164.473,Z 360.462,A -85,B 0,C 180,E1 -24061.859,E2 -24061.859} C_VEL
LIN {X 0,Y 158.043,Z 349.425,A -85,B 0,C 180,E1 -24064.365,E2 -24064.365} C_VEL
LIN {X 0,Y 154.708,Z 344.598,A -85,B 0,C 180,E1 -24065.73,E2 -24065.73} C_VEL
LIN {X 0,Y 152.669,Z 341.324,A -85,B 0,C 180,E1 -24066.629,E2 -24066.629} C_VEL
LIN {X 0,Y 150.772,Z 338.876,A -85,B 0,C 180,E1 -24067.458,E2 -24067.458} C_VEL
LIN {X 0,Y 150.168,Z 336.78,A -85,B 0,C 180,E1 -24067.895,E2 -24067.895} C_VEL
LIN {X 0,Y 150.129,Z 336.772,A -85,B 0,C 180,E1 -24071.494,E2 -24071.494} C_VEL
LIN {X 0,Y 150.123,Z 336.774,A -85,B 0,C 180,E1 -24075.393,E2 -24075.393} C_VEL
LIN {X 0,Y 150.132,Z 336.773,A -85,B 0,C 180,E1 -24079.051,E2 -24079.051} C_VEL
LIN {X 0,Y 150.171,Z 336.765,A -85,B 0,C 180,E1 -24082.708,E2 -24082.708} C_VEL
LIN {X 0,Y 150.203,Z 336.763,A -85,B 0,C 180,E1 -24087.37,E2 -24087.37} C_VEL
LIN {X 0,Y 150.179,Z 336.752,A -85,B 0,C 180,E1 -24092.761,E2 -24092.761} C_VEL
LIN {X 0,Y 150.276,Z 336.766,A -85,B 0,C 180,E1 -24099.277,E2 -24099.277} C_VEL
LIN {X 0,Y 150.301,Z 336.732,A -85,B 0,C 180,E1 -24103.706,E2 -24103.706} C_VEL
LIN {X 0,Y 150.598,Z 336.724,A -85,B 0,C 180,E1 -24109.241,E2 -24109.241} C_VEL
LIN {X 0,Y 150.672,Z 336.708,A -85,B 0,C 180,E1 -24111.955,E2 -24111.955} C_VEL
LIN {X 0,Y 151.19,Z 336.65,A -85,B 0,C 180,E1 -24119.999,E2 -24119.999} C_VEL
LIN {X 0,Y 150.692,Z 336.698,A -85,B 0,C 180,E1 -24128.042,E2 -24128.042} C_VEL
LIN {X 0,Y 150.568,Z 336.728,A -85,B 0,C 180,E1 -24131.431,E2 -24131.431} C_VEL
LIN {X 0,Y 150.321,Z 336.734,A -85,B 0,C 180,E1 -24136.291,E2 -24136.291} C_VEL
LIN {X 0,Y 150.333,Z 336.759,A -85,B 0,C 180,E1 -24140.78,E2 -24140.78} C_VEL
LIN {X 0,Y 150.235,Z 336.764,A -85,B 0,C 180,E1 -24147.28,E2 -24147.28} C_VEL
LIN {X 0,Y 150.208,Z 336.767,A -85,B 0,C 180,E1 -24152.632,E2 -24152.632} C_VEL
LIN {X 0,Y 150.163,Z 336.774,A -85,B 0,C 180,E1 -24157.476,E2 -24157.476} C_VEL
LIN {X 0,Y 150.174,Z 336.871,A -85,B 0,C 180,E1 -24160.822,E2 -24160.822} C_VEL
LIN {X 0,Y 151.112,Z 339.575,A -85,B 0,C 180,E1 -24161.34,E2 -24161.34} C_VEL
LIN {X 0,Y 153.195,Z 342.057,A -85,B 0,C 180,E1 -24162.233,E2 -24162.233} C_VEL
LIN {X 0,Y 155.363,Z 345.41,A -85,B 0,C 180,E1 -24163.172,E2 -24163.172} C_VEL
LIN {X 0,Y 158.375,Z 350.556,A -85,B 0,C 180,E1 -24164.44,E2 -24164.44} C_VEL
LIN {X 0,Y 163.885,Z 361.666,A -85,B 0,C 180,E1 -24166.678,E2 -24166.678} C_VEL
LIN {X 0,Y 168.899,Z 373.944,A -85,B 0,C 180,E1 -24168.648,E2 -24168.648} C_VEL
LIN {X 0,Y 172.033,Z 382.828,A -85,B 0,C 180,E1 -24169.86,E2 -24169.86} C_VEL
LIN {X 0,Y 173.149,Z 396.536,A -85,B 0,C 180,E1 -24170.8,E2 -24170.8} C_VEL
LIN {X 0,Y 170.542,Z 444.35,A -85,B 0,C 180,E1 -24172.662,E2 -24172.662} C_VEL
LIN {X 0,Y 169.098,Z 457.591,A -85,B 0,C 180,E1 -24173.593,E2 -24173.593} C_VEL
LIN {X 0,Y 167.076,Z 469.731,A -85,B 0,C 180,E1 -24174.85,E2 -24174.85} C_VEL
LIN {X 0,Y 164.844,Z 480.308,A -85,B 0,C 180,E1 -24176.344,E2 -24176.344} C_VEL
LIN {X 0,Y 161.784,Z 492.276,A -85,B 0,C 180,E1 -24178.584,E2 -24178.584} C_VEL
LIN {X 0,Y 158.755,Z 502.961,A -85,B 0,C 180,E1 -24181.224,E2 -24181.224} C_VEL
LIN {X 0,Y 155.795,Z 513.025,A -85,B 0,C 180,E1 -24184.45,E2 -24184.45} C_VEL
LIN {X 0,Y 153.283,Z 521.145,A -85,B 0,C 180,E1 -24187.776,E2 -24187.776} C_VEL
LIN {X 0,Y 150.933,Z 528.683,A -85,B 0,C 180,E1 -24191.683,E2 -24191.683} C_VEL
LIN {X 0,Y 149.003,Z 535.623,A -85,B 0,C 180,E1 -24196.361,E2 -24196.361} C_VEL
LIN {X 0,Y 148.235,Z 539.434,A -85,B 0,C 180,E1 -24199.717,E2 -24199.717} C_VEL
LIN {X 0,Y 147.285,Z 541.485,A -85,B 0,C 180,E1 -24201.834,E2 -24201.834} C_VEL
LIN {X 0,Y 145.581,Z 543.222,A -85,B 0,C 180,E1 -24203.956,E2 -24203.956} C_VEL
LIN {X 0,Y 141.82,Z 545.791,A -85,B 0,C 180,E1 -24208.383,E2 -24208.383} C_VEL
LIN {X 0,Y 140.595,Z 546.898,A -85,B 0,C 180,E1 -24211.553,E2 -24211.553} C_VEL
LIN {X 0,Y 140.62,Z 547.769,A -85,B 0,C 180,E1 -24215.739,E2 -24215.739} C_VEL
LIN {X 0,Y 140.906,Z 547.861,A -85,B 0,C 180,E1 -24218.608,E2 -24218.608} C_VEL
LIN {X 0,Y 142.335,Z 546.887,A -85,B 0,C 180,E1 -24224.295,E2 -24224.295} C_VEL
LIN {X 0,Y 143.509,Z 545.832,A -85,B 0,C 180,E1 -24227.09,E2 -24227.09} C_VEL
LIN {X 0,Y 145.047,Z 544.357,A -85,B 0,C 180,E1 -24229.828,E2 -24229.828} C_VEL
LIN {X 0,Y 148.076,Z 541.361,A -85,B 0,C 180,E1 -24233.795,E2 -24233.795} C_VEL
LIN {X 0,Y 151.731,Z 537.337,A -85,B 0,C 180,E1 -24237.595,E2 -24237.595} C_VEL
LIN {X 0,Y 156.677,Z 531.184,A -85,B 0,C 180,E1 -24241.808,E2 -24241.808} C_VEL
LIN {X 0,Y 161.589,Z 524.505,A -85,B 0,C 180,E1 -24245.191,E2 -24245.191} C_VEL
LIN {X 0,Y 167.223,Z 516.237,A -85,B 0,C 180,E1 -24248.311,E2 -24248.311} C_VEL
LIN {X 0,Y 172.256,Z 507.766,A -85,B 0,C 180,E1 -24250.754,E2 -24250.754} C_VEL
LIN {X 0,Y 177.605,Z 497.328,A -85,B 0,C 180,E1 -24253.049,E2 -24253.049} C_VEL
LIN {X 0,Y 182.121,Z 487.016,A -85,B 0,C 180,E1 -24254.772,E2 -24254.772} C_VEL
LIN {X 0,Y 186.259,Z 475.722,A -85,B 0,C 180,E1 -24256.191,E2 -24256.191} C_VEL
LIN {X 0,Y 189.57,Z 464.179,A -85,B 0,C 180,E1 -24257.268,E2 -24257.268} C_VEL
LIN {X 0,Y 192.371,Z 450.598,A -85,B 0,C 180,E1 -24258.145,E2 -24258.145} C_VEL
LIN {X 0,Y 194.004,Z 437.11,A -85,B 0,C 180,E1 -24258.71,E2 -24258.71} C_VEL
LIN {X 0,Y 195.708,Z 415.419,A -85,B 0,C 180,E1 -24259.362,E2 -24259.362} C_VEL
LIN {X 0,Y 193.262,Z 408.642,A -85,B 0,C 180,E1 -24260.814,E2 -24260.814} C_VEL
LIN {X 0,Y 188.865,Z 398.574,A -85,B 0,C 180,E1 -24263.523,E2 -24263.523} C_VEL
LIN {X 0,Y 184.358,Z 389.603,A -85,B 0,C 180,E1 -24266.594,E2 -24266.594} C_VEL
LIN {X 0,Y 179.946,Z 381.48,A -85,B 0,C 180,E1 -24270.051,E2 -24270.051} C_VEL
LIN {X 0,Y 177.139,Z 376.838,A -85,B 0,C 180,E1 -24272.554,E2 -24272.554} C_VEL
LIN {X 0,Y 174.339,Z 372.278,A -85,B 0,C 180,E1 -24275.436,E2 -24275.436} C_VEL
LIN {X 0,Y 171.804,Z 369.227,A -85,B 0,C 180,E1 -24278.398,E2 -24278.398} C_VEL
LIN {X 0,Y 170.813,Z 367.433,A -85,B 0,C 180,E1 -24279.844,E2 -24279.844} C_VEL
LIN {X 0,Y 168.212,Z 364.853,A -85,B 0,C 180,E1 -24284.197,E2 -24284.197} C_VEL
LIN {X 0,Y 167.125,Z 362.112,A -85,B 0,C 180,E1 -24287.246,E2 -24287.246} C_VEL
LIN {X 0,Y 165.865,Z 361.419,A -85,B 0,C 180,E1 -24292.698,E2 -24292.698} C_VEL
LIN {X 0,Y 166.481,Z 361.485,A -85,B 0,C 180,E1 -24300,E2 -24300} C_VEL
LIN {X 0,Y 167.338,Z 362.147,A -85,B 0,C 180,E1 -24302.719,E2 -24302.719} C_VEL
LIN {X 0,Y 168.93,Z 365.456,A -85,B 0,C 180,E1 -24306.578,E2 -24306.578} C_VEL
LIN {X 0,Y 171.133,Z 367.687,A -85,B 0,C 180,E1 -24310.015,E2 -24310.015} C_VEL
LIN {X 0,Y 173.387,Z 371.237,A -85,B 0,C 180,E1 -24312.956,E2 -24312.956} C_VEL
LIN {X 0,Y 174.683,Z 372.578,A -85,B 0,C 180,E1 -24314.341,E2 -24314.341} C_VEL
LIN {X 0,Y 177.386,Z 376.485,A -85,B 0,C 180,E1 -24317.027,E2 -24317.027} C_VEL
LIN {X 0,Y 181.312,Z 382.143,A -85,B 0,C 180,E1 -24320.344,E2 -24320.344} C_VEL
LIN {X 0,Y 185.658,Z 388.738,A -85,B 0,C 180,E1 -24323.495,E2 -24323.495} C_VEL
LIN {X 0,Y 191.091,Z 397.88,A -85,B 0,C 180,E1 -24326.919,E2 -24326.919} C_VEL
LIN {X 0,Y 195.198,Z 406.667,A -85,B 0,C 180,E1 -24329.307,E2 -24329.307} C_VEL
LIN {X 0,Y 196.127,Z 408.885,A -85,B 0,C 180,E1 -24329.829,E2 -24329.829} C_VEL
LIN {X 0,Y 193.663,Z 437.948,A -85,B 0,C 180,E1 -24330.753,E2 -24330.753} C_VEL
LIN {X 0,Y 191.374,Z 451.687,A -85,B 0,C 180,E1 -24331.501,E2 -24331.501} C_VEL
LIN {X 0,Y 188.536,Z 463.592,A -85,B 0,C 180,E1 -24332.499,E2 -24332.499} C_VEL
LIN {X 0,Y 185.035,Z 474.876,A -85,B 0,C 180,E1 -24333.811,E2 -24333.811} C_VEL
LIN {X 0,Y 180.539,Z 486.574,A -85,B 0,C 180,E1 -24335.635,E2 -24335.635} C_VEL
LIN {X 0,Y 175.584,Z 497.088,A -85,B 0,C 180,E1 -24337.764,E2 -24337.764} C_VEL
LIN {X 0,Y 170.37,Z 506.439,A -85,B 0,C 180,E1 -24340.255,E2 -24340.255} C_VEL
LIN {X 0,Y 165.848,Z 513.591,A -85,B 0,C 180,E1 -24342.69,E2 -24342.69} C_VEL
LIN {X 0,Y 160.064,Z 521.603,A -85,B 0,C 180,E1 -24346.246,E2 -24346.246} C_VEL
LIN {X 0,Y 156.082,Z 526.649,A -85,B 0,C 180,E1 -24349.237,E2 -24349.237} C_VEL
LIN {X 0,Y 151.8,Z 531.507,A -85,B 0,C 180,E1 -24352.994,E2 -24352.994} C_VEL
LIN {X 0,Y 148.217,Z 535.194,A -85,B 0,C 180,E1 -24356.953,E2 -24356.953} C_VEL
LIN {X 0,Y 145.322,Z 537.815,A -85,B 0,C 180,E1 -24361.076,E2 -24361.076} C_VEL
LIN {X 0,Y 143.744,Z 539.031,A -85,B 0,C 180,E1 -24363.892,E2 -24363.892} C_VEL
LIN {X 0,Y 142.491,Z 539.791,A -85,B 0,C 180,E1 -24366.758,E2 -24366.758} C_VEL
LIN {X 0,Y 141.246,Z 540.182,A -85,B 0,C 180,E1 -24370.979,E2 -24370.979} C_VEL
LIN {X 0,Y 140.455,Z 539.635,A -85,B 0,C 180,E1 -24375.509,E2 -24375.509} C_VEL
LIN {X 0,Y 140.255,Z 538.74,A -85,B 0,C 180,E1 -24378.436,E2 -24378.436} C_VEL
LIN {X 0,Y 140.291,Z 537.444,A -85,B 0,C 180,E1 -24381.354,E2 -24381.354} C_VEL
LIN {X 0,Y 140.907,Z 534.488,A -85,B 0,C 180,E1 -24385.993,E2 -24385.993} C_VEL
LIN {X 0,Y 141.651,Z 530.96,A -85,B 0,C 180,E1 -24389.998,E2 -24389.998} C_VEL
LIN {X 0,Y 142.964,Z 526.102,A -85,B 0,C 180,E1 -24394.227,E2 -24394.227} C_VEL
LIN {X 0,Y 144.862,Z 519.984,A -85,B 0,C 180,E1 -24398.367,E2 -24398.367} C_VEL
LIN {X 0,Y 147.464,Z 512.373,A -85,B 0,C 180,E1 -24402.382,E2 -24402.382} C_VEL
LIN {X 0,Y 150.025,Z 504.592,A -85,B 0,C 180,E1 -24405.624,E2 -24405.624} C_VEL
LIN {X 0,Y 153.459,Z 493.998,A -85,B 0,C 180,E1 -24409.042,E2 -24409.042} C_VEL
LIN {X 0,Y 156.802,Z 483.171,A -85,B 0,C 180,E1 -24411.699,E2 -24411.699} C_VEL
LIN {X 0,Y 159.321,Z 472.68,A -85,B 0,C 180,E1 -24413.734,E2 -24413.734} C_VEL
LIN {X 0,Y 161.816,Z 460.064,A -85,B 0,C 180,E1 -24415.567,E2 -24415.567} C_VEL
LIN {X 0,Y 163.662,Z 447.484,A -85,B 0,C 180,E1 -24416.885,E2 -24416.885} C_VEL
LIN {X 0,Y 164.957,Z 434.158,A -85,B 0,C 180,E1 -24417.772,E2 -24417.772} C_VEL
LIN {X 0,Y 167.92,Z 382.832,A -85,B 0,C 180,E1 -24419.764,E2 -24419.764} C_VEL
LIN {X 0,Y 165.277,Z 375.857,A -85,B 0,C 180,E1 -24420.809,E2 -24420.809} C_VEL
LIN {X 0,Y 158.802,Z 362.924,A -85,B 0,C 180,E1 -24423.344,E2 -24423.344} C_VEL
LIN {X 0,Y 153.129,Z 353.443,A -85,B 0,C 180,E1 -24425.711,E2 -24425.711} C_VEL
LIN {X 0,Y 148.459,Z 346.347,A -85,B 0,C 180,E1 -24427.818,E2 -24427.818} C_VEL
LIN {X 0,Y 146.342,Z 343.105,A -85,B 0,C 180,E1 -24428.845,E2 -24428.845} C_VEL
LIN {X 0,Y 143.746,Z 339.89,A -85,B 0,C 180,E1 -24430.118,E2 -24430.118} C_VEL
LIN {X 0,Y 143.085,Z 337.648,A -85,B 0,C 180,E1 -24430.579,E2 -24430.579} C_VEL
LIN {X 0,Y 143.029,Z 337.649,A -85,B 0,C 180,E1 -24436.534,E2 -24436.534} C_VEL
LIN {X 0,Y 143.068,Z 337.658,A -85,B 0,C 180,E1 -24441.807,E2 -24441.807} C_VEL
LIN {X 0,Y 143.171,Z 337.638,A -85,B 0,C 180,E1 -24447.318,E2 -24447.318} C_VEL
LIN {X 0,Y 143.1,Z 337.628,A -85,B 0,C 180,E1 -24453.767,E2 -24453.767} C_VEL
LIN {X 0,Y 143.239,Z 337.642,A -85,B 0,C 180,E1 -24459.912,E2 -24459.912} C_VEL
LIN {X 0,Y 143.295,Z 337.605,A -85,B 0,C 180,E1 -24465.804,E2 -24465.804} C_VEL
LIN {X 0,Y 143.525,Z 337.603,A -85,B 0,C 180,E1 -24468.704,E2 -24468.704} C_VEL
LIN {X 0,Y 143.598,Z 337.591,A -85,B 0,C 180,E1 -24471.556,E2 -24471.556} C_VEL
LIN {X 0,Y 144.148,Z 337.527,A -85,B 0,C 180,E1 -24479.999,E2 -24479.999} C_VEL
LIN {X 0,Y 143.614,Z 337.583,A -85,B 0,C 180,E1 -24488.442,E2 -24488.442} C_VEL
LIN {X 0,Y 143.494,Z 337.609,A -85,B 0,C 180,E1 -24491.62,E2 -24491.62} C_VEL
LIN {X 0,Y 143.261,Z 337.617,A -85,B 0,C 180,E1 -24497.118,E2 -24497.118} C_VEL
LIN {X 0,Y 143.261,Z 337.637,A -85,B 0,C 180,E1 -24501.245,E2 -24501.245} C_VEL
LIN {X 0,Y 143.182,Z 337.64,A -85,B 0,C 180,E1 -24507.936,E2 -24507.936} C_VEL
LIN {X 0,Y 143.136,Z 337.647,A -85,B 0,C 180,E1 -24513.42,E2 -24513.42} C_VEL
LIN {X 0,Y 143.099,Z 337.664,A -85,B 0,C 180,E1 -24518.082,E2 -24518.082} C_VEL
LIN {X 0,Y 143.99,Z 340.283,A -85,B 0,C 180,E1 -24518.643,E2 -24518.643} C_VEL
LIN {X 0,Y 146.332,Z 343.137,A -85,B 0,C 180,E1 -24519.783,E2 -24519.783} C_VEL
LIN {X 0,Y 148.52,Z 346.471,A -85,B 0,C 180,E1 -24520.843,E2 -24520.843} C_VEL
LIN {X 0,Y 153.364,Z 353.91,A -85,B 0,C 180,E1 -24523.031,E2 -24523.031} C_VEL
LIN {X 0,Y 159.36,Z 366.431,A -85,B 0,C 180,E1 -24525.658,E2 -24525.658} C_VEL
LIN {X 0,Y 164.208,Z 378.785,A -85,B 0,C 180,E1 -24527.699,E2 -24527.699} C_VEL
LIN {X 0,Y 166.345,Z 384.959,A -85,B 0,C 180,E1 -24528.584,E2 -24528.584} C_VEL
LIN {X 0,Y 167.295,Z 397.116,A -85,B 0,C 180,E1 -24529.458,E2 -24529.458} C_VEL
LIN {X 0,Y 164.57,Z 444.461,A -85,B 0,C 180,E1 -24531.352,E2 -24531.352} C_VEL
LIN {X 0,Y 163.038,Z 457.824,A -85,B 0,C 180,E1 -24532.327,E2 -24532.327} C_VEL
LIN {X 0,Y 160.865,Z 470.258,A -85,B 0,C 180,E1 -24533.666,E2 -24533.666} C_VEL
LIN {X 0,Y 158.18,Z 482.298,A -85,B 0,C 180,E1 -24535.497,E2 -24535.497} C_VEL
LIN {X 0,Y 154.963,Z 493.799,A -85,B 0,C 180,E1 -24537.801,E2 -24537.801} C_VEL
LIN {X 0,Y 151.811,Z 504.178,A -85,B 0,C 180,E1 -24540.539,E2 -24540.539} C_VEL
LIN {X 0,Y 148.716,Z 514.074,A -85,B 0,C 180,E1 -24543.969,E2 -24543.969} C_VEL
LIN {X 0,Y 146.719,Z 520.488,A -85,B 0,C 180,E1 -24546.725,E2 -24546.725} C_VEL
LIN {X 0,Y 144.176,Z 528.106,A -85,B 0,C 180,E1 -24550.792,E2 -24550.792} C_VEL
LIN {X 0,Y 142.08,Z 535.134,A -85,B 0,C 180,E1 -24555.683,E2 -24555.683} C_VEL
LIN {X 0,Y 141.082,Z 539.768,A -85,B 0,C 180,E1 -24559.961,E2 -24559.961} C_VEL
LIN {X 0,Y 140.619,Z 543.273,A -85,B 0,C 180,E1 -24564.265,E2 -24564.265} C_VEL
LIN {X 0,Y 140.595,Z 545.82,A -85,B 0,C 180,E1 -24568.713,E2 -24568.713} C_VEL
LIN {X 0,Y 140.595,Z 546.898,A -85,B 0,C 180,E1 -24571.553,E2 -24571.553} C_VEL
LIN {X 0,Y 139.853,Z 547.463,A -85,B 0,C 180,E1 -24573.937,E2 -24573.937} C_VEL
LIN {X 0,Y 137.226,Z 547.761,A -85,B 0,C 180,E1 -24577.89,E2 -24577.89} C_VEL
LIN {X 0,Y 135.376,Z 547.56,A -85,B 0,C 180,E1 -24581.154,E2 -24581.154} C_VEL
LIN {X 0,Y 135.113,Z 547.024,A -85,B 0,C 180,E1 -24584.08,E2 -24584.08} C_VEL
LIN {X 0,Y 135.238,Z 546.876,A -85,B 0,C 180,E1 -24584.495,E2 -24584.495} C_VEL
LIN {X 0,Y 136.703,Z 545.728,A -85,B 0,C 180,E1 -24587.969,E2 -24587.969} C_VEL
LIN {X 0,Y 138.382,Z 544.306,A -85,B 0,C 180,E1 -24590.827,E2 -24590.827} C_VEL
LIN {X 0,Y 141.584,Z 541.356,A -85,B 0,C 180,E1 -24594.958,E2 -24594.958} C_VEL
LIN {X 0,Y 145.477,Z 537.388,A -85,B 0,C 180,E1 -24598.89,E2 -24598.89} C_VEL
LIN {X 0,Y 149.891,Z 532.314,A -85,B 0,C 180,E1 -24602.63,E2 -24602.63} C_VEL
LIN {X 0,Y 154.924,Z 525.955,A -85,B 0,C 180,E1 -24606.14,E2 -24606.14} C_VEL
LIN {X 0,Y 160.715,Z 518.029,A -85,B 0,C 180,E1 -24609.353,E2 -24609.353} C_VEL
LIN {X 0,Y 165.91,Z 509.977,A -85,B 0,C 180,E1 -24611.851,E2 -24611.851} C_VEL
LIN {X 0,Y 171.396,Z 500.177,A -85,B 0,C 180,E1 -24614.195,E2 -24614.195} C_VEL
LIN {X 0,Y 176.583,Z 489.226,A -85,B 0,C 180,E1 -24616.17,E2 -24616.17} C_VEL
LIN {X 0,Y 180.838,Z 478.505,A -85,B 0,C 180,E1 -24617.598,E2 -24617.598} C_VEL
LIN {X 0,Y 184.878,Z 465.607,A -85,B 0,C 180,E1 -24618.866,E2 -24618.866} C_VEL
LIN {X 0,Y 187.796,Z 452.648,A -85,B 0,C 180,E1 -24619.76,E2 -24619.76} C_VEL
LIN {X 0,Y 189.71,Z 438.896,A -85,B 0,C 180,E1 -24620.361,E2 -24620.361} C_VEL
LIN {X 0,Y 191.359,Z 417.431,A -85,B 0,C 180,E1 -24621.07,E2 -24621.07} C_VEL
LIN {X 0,Y 187.373,Z 407.313,A -85,B 0,C 180,E1 -24623.633,E2 -24623.633} C_VEL
LIN {X 0,Y 183.317,Z 398.468,A -85,B 0,C 180,E1 -24626.475,E2 -24626.475} C_VEL
LIN {X 0,Y 179.544,Z 390.932,A -85,B 0,C 180,E1 -24629.449,E2 -24629.449} C_VEL
LIN {X 0,Y 177.209,Z 386.609,A -85,B 0,C 180,E1 -24631.502,E2 -24631.502} C_VEL
LIN {X 0,Y 174.879,Z 382.576,A -85,B 0,C 180,E1 -24633.765,E2 -24633.765} C_VEL
LIN {X 0,Y 172.685,Z 378.859,A -85,B 0,C 180,E1 -24636.184,E2 -24636.184} C_VEL
LIN {X 0,Y 170.11,Z 375.448,A -85,B 0,C 180,E1 -24639.441,E2 -24639.441} C_VEL
LIN {X 0,Y 169.358,Z 374.173,A -85,B 0,C 180,E1 -24640.611,E2 -24640.611} C_VEL
LIN {X 0,Y 166.894,Z 371.377,A -85,B 0,C 180,E1 -24645.147,E2 -24645.147} C_VEL
LIN {X 0,Y 166.058,Z 369.057,A -85,B 0,C 180,E1 -24647.784,E2 -24647.784} C_VEL
LIN {X 0,Y 164.887,Z 368.436,A -85,B 0,C 180,E1 -24655.11,E2 -24655.11} C_VEL
LIN {X 0,Y 165.764,Z 368.666,A -85,B 0,C 180,E1 -24660.608,E2 -24660.608} C_VEL
LIN {X 0,Y 166.296,Z 369.158,A -85,B 0,C 180,E1 -24662.309,E2 -24662.309} C_VEL
LIN {X 0,Y 167.88,Z 372.452,A -85,B 0,C 180,E1 -24666.31,E2 -24666.31} C_VEL
LIN {X 0,Y 169.713,Z 374.364,A -85,B 0,C 180,E1 -24669.31,E2 -24669.31} C_VEL
LIN {X 0,Y 172.096,Z 378.141,A -85,B 0,C 180,E1 -24672.567,E2 -24672.567} C_VEL
LIN {X 0,Y 173.161,Z 379.41,A -85,B 0,C 180,E1 -24673.766,E2 -24673.766} C_VEL
LIN {X 0,Y 176.612,Z 384.51,A -85,B 0,C 180,E1 -24677.26,E2 -24677.26} C_VEL
LIN {X 0,Y 179.391,Z 388.773,A -85,B 0,C 180,E1 -24679.675,E2 -24679.675} C_VEL
LIN {X 0,Y 183.437,Z 395.163,A -85,B 0,C 180,E1 -24682.751,E2 -24682.751} C_VEL
LIN {X 0,Y 188.33,Z 403.721,A -85,B 0,C 180,E1 -24686.008,E2 -24686.008} C_VEL
LIN {X 0,Y 191.808,Z 411.583,A -85,B 0,C 180,E1 -24688.168,E2 -24688.168} C_VEL
LIN {X 0,Y 189.634,Z 437.341,A -85,B 0,C 180,E1 -24689.009,E2 -24689.009} C_VEL
LIN {X 0,Y 187.286,Z 451.055,A -85,B 0,C 180,E1 -24689.714,E2 -24689.714} C_VEL
LIN {X 0,Y 184.435,Z 463.036,A -85,B 0,C 180,E1 -24690.709,E2 -24690.709} C_VEL
LIN {X 0,Y 181.045,Z 473.671,A -85,B 0,C 180,E1 -24691.877,E2 -24691.877} C_VEL
LIN {X 0,Y 176.926,Z 484.352,A -85,B 0,C 180,E1 -24693.468,E2 -24693.468} C_VEL
LIN {X 0,Y 171.776,Z 495.283,A -85,B 0,C 180,E1 -24695.592,E2 -24695.592} C_VEL
LIN {X 0,Y 166.802,Z 504.159,A -85,B 0,C 180,E1 -24697.812,E2 -24697.812} C_VEL
LIN {X 0,Y 161.684,Z 512.135,A -85,B 0,C 180,E1 -24700.378,E2 -24700.378} C_VEL
LIN {X 0,Y 155.811,Z 520.178,A -85,B 0,C 180,E1 -24703.803,E2 -24703.803} C_VEL
LIN {X 0,Y 150.575,Z 526.45,A -85,B 0,C 180,E1 -24707.405,E2 -24707.405} C_VEL
LIN {X 0,Y 146.018,Z 531.394,A -85,B 0,C 180,E1 -24711.264,E2 -24711.264} C_VEL
LIN {X 0,Y 142.1,Z 535.161,A -85,B 0,C 180,E1 -24715.334,E2 -24715.334} C_VEL
LIN {X 0,Y 138.943,Z 537.858,A -85,B 0,C 180,E1 -24719.612,E2 -24719.612} C_VEL
LIN {X 0,Y 137.197,Z 539.111,A -85,B 0,C 180,E1 -24722.544,E2 -24722.544} C_VEL
LIN {X 0,Y 135.797,Z 539.941,A -85,B 0,C 180,E1 -24725.54,E2 -24725.54} C_VEL
LIN {X 0,Y 133.978,Z 540.303,A -85,B 0,C 180,E1 -24731.653,E2 -24731.653} C_VEL
LIN {X 0,Y 133.451,Z 539.896,A -85,B 0,C 180,E1 -24734.731,E2 -24734.731} C_VEL
LIN {X 0,Y 133.169,Z 539.066,A -85,B 0,C 180,E1 -24737.811,E2 -24737.811} C_VEL
LIN {X 0,Y 133.179,Z 537.803,A -85,B 0,C 180,E1 -24740.889,E2 -24740.889} C_VEL
LIN {X 0,Y 133.835,Z 534.649,A -85,B 0,C 180,E1 -24746.157,E2 -24746.157} C_VEL
LIN {X 0,Y 134.866,Z 530.032,A -85,B 0,C 180,E1 -24751.491,E2 -24751.491} C_VEL
LIN {X 0,Y 136.762,Z 523.847,A -85,B 0,C 180,E1 -24756.637,E2 -24756.637} C_VEL
LIN {X 0,Y 139.112,Z 517.112,A -85,B 0,C 180,E1 -24760.918,E2 -24760.918} C_VEL
LIN {X 0,Y 142.103,Z 508.755,A -85,B 0,C 180,E1 -24765.047,E2 -24765.047} C_VEL
LIN {X 0,Y 145.064,Z 500.144,A -85,B 0,C 180,E1 -24768.353,E2 -24768.353} C_VEL
LIN {X 0,Y 148.257,Z 490.679,A -85,B 0,C 180,E1 -24771.187,E2 -24771.187} C_VEL
LIN {X 0,Y 151.367,Z 480.357,A -85,B 0,C 180,E1 -24773.605,E2 -24773.605} C_VEL
LIN {X 0,Y 154.109,Z 469.104,A -85,B 0,C 180,E1 -24775.671,E2 -24775.671} C_VEL
LIN {X 0,Y 156.299,Z 457.68,A -85,B 0,C 180,E1 -24777.261,E2 -24777.261} C_VEL
LIN {X 0,Y 158.152,Z 444.596,A -85,B 0,C 180,E1 -24778.534,E2 -24778.534} C_VEL
LIN {X 0,Y 159.4,Z 430.818,A -85,B 0,C 180,E1 -24779.355,E2 -24779.355} C_VEL
LIN {X 0,Y 162.104,Z 384.403,A -85,B 0,C 180,E1 -24781.19,E2 -24781.19} C_VEL
LIN {X 0,Y 159.369,Z 377.646,A -85,B 0,C 180,E1 -24782.332,E2 -24782.332} C_VEL
LIN {X 0,Y 152.932,Z 364.968,A -85,B 0,C 180,E1 -24785.062,E2 -24785.062} C_VEL
LIN {X 0,Y 146.592,Z 354.661,A -85,B 0,C 180,E1 -24787.964,E2 -24787.964} C_VEL
LIN {X 0,Y 144.054,Z 350.867,A -85,B 0,C 180,E1 -24789.216,E2 -24789.216} C_VEL
LIN {X 0,Y 141.716,Z 347.468,A -85,B 0,C 180,E1 -24790.429,E2 -24790.429} C_VEL
LIN {X 0,Y 139.501,Z 344.141,A -85,B 0,C 180,E1 -24791.65,E2 -24791.65} C_VEL
LIN {X 0,Y 138.273,Z 342.923,A -85,B 0,C 180,E1 -24792.309,E2 -24792.309} C_VEL
LIN {X 0,Y 136.571,Z 340.555,A -85,B 0,C 180,E1 -24793.31,E2 -24793.31} C_VEL
LIN {X 0,Y 135.992,Z 338.545,A -85,B 0,C 180,E1 -24793.842,E2 -24793.842} C_VEL
LIN {X 0,Y 135.978,Z 338.526,A -85,B 0,C 180,E1 -24797.785,E2 -24797.785} C_VEL
LIN {X 0,Y 136.017,Z 338.537,A -85,B 0,C 180,E1 -24801.68,E2 -24801.68} C_VEL
LIN {X 0,Y 136.048,Z 338.511,A -85,B 0,C 180,E1 -24805.74,E2 -24805.74} C_VEL
LIN {X 0,Y 136.057,Z 338.523,A -85,B 0,C 180,E1 -24811.412,E2 -24811.412} C_VEL
LIN {X 0,Y 136.175,Z 338.522,A -85,B 0,C 180,E1 -24818.821,E2 -24818.821} C_VEL
LIN {X 0,Y 136.214,Z 338.483,A -85,B 0,C 180,E1 -24825.049,E2 -24825.049} C_VEL
LIN {X 0,Y 136.419,Z 338.484,A -85,B 0,C 180,E1 -24828.177,E2 -24828.177} C_VEL
LIN {X 0,Y 136.528,Z 338.475,A -85,B 0,C 180,E1 -24831.116,E2 -24831.116} C_VEL
LIN {X 0,Y 137.105,Z 338.404,A -85,B 0,C 180,E1 -24839.999,E2 -24839.999} C_VEL
LIN {X 0,Y 136.54,Z 338.467,A -85,B 0,C 180,E1 -24848.882,E2 -24848.882} C_VEL
LIN {X 0,Y 136.409,Z 338.491,A -85,B 0,C 180,E1 -24851.893,E2 -24851.893} C_VEL
LIN {X 0,Y 136.181,Z 338.507,A -85,B 0,C 180,E1 -24858.037,E2 -24858.037} C_VEL
LIN {X 0,Y 136.184,Z 338.516,A -85,B 0,C 180,E1 -24861.74,E2 -24861.74} C_VEL
LIN {X 0,Y 136.093,Z 338.522,A -85,B 0,C 180,E1 -24868.615,E2 -24868.615} C_VEL
LIN {X 0,Y 136.04,Z 338.538,A -85,B 0,C 180,E1 -24874.854,E2 -24874.854} C_VEL
LIN {X 0,Y 136.988,Z 341.305,A -85,B 0,C 180,E1 -24875.589,E2 -24875.589} C_VEL
LIN {X 0,Y 139.49,Z 344.068,A -85,B 0,C 180,E1 -24876.974,E2 -24876.974} C_VEL
LIN {X 0,Y 141.652,Z 347.418,A -85,B 0,C 180,E1 -24878.172,E2 -24878.172} C_VEL
LIN {X 0,Y 143.1,Z 349.48,A -85,B 0,C 180,E1 -24878.928,E2 -24878.928} C_VEL
LIN {X 0,Y 148.127,Z 357.043,A -85,B 0,C 180,E1 -24881.397,E2 -24881.397} C_VEL
LIN {X 0,Y 152.949,Z 366.709,A -85,B 0,C 180,E1 -24883.684,E2 -24883.684} C_VEL
LIN {X 0,Y 158.077,Z 379.423,A -85,B 0,C 180,E1 -24886.028,E2 -24886.028} C_VEL
LIN {X 0,Y 160.861,Z 388.036,A -85,B 0,C 180,E1 -24887.304,E2 -24887.304} C_VEL
LIN {X 0,Y 161.552,Z 397.783,A -85,B 0,C 180,E1 -24888.029,E2 -24888.029} C_VEL
LIN {X 0,Y 158.751,Z 444.035,A -85,B 0,C 180,E1 -24889.915,E2 -24889.915} C_VEL
LIN {X 0,Y 157.161,Z 457.364,A -85,B 0,C 180,E1 -24890.9,E2 -24890.9} C_VEL
LIN {X 0,Y 154.943,Z 469.652,A -85,B 0,C 180,E1 -24892.244,E2 -24892.244} C_VEL
LIN {X 0,Y 152.305,Z 481.003,A -85,B 0,C 180,E1 -24893.964,E2 -24893.964} C_VEL
LIN {X 0,Y 148.99,Z 492.717,A -85,B 0,C 180,E1 -24896.343,E2 -24896.343} C_VEL
LIN {X 0,Y 145.682,Z 503.259,A -85,B 0,C 180,E1 -24899.167,E2 -24899.167} C_VEL
LIN {X 0,Y 142.88,Z 511.838,A -85,B 0,C 180,E1 -24902.126,E2 -24902.126} C_VEL
LIN {X 0,Y 140.207,Z 519.816,A -85,B 0,C 180,E1 -24905.575,E2 -24905.575} C_VEL
LIN {X 0,Y 137.436,Z 527.522,A -85,B 0,C 180,E1 -24909.81,E2 -24909.81} C_VEL
LIN {X 0,Y 135.663,Z 532.79,A -85,B 0,C 180,E1 -24913.448,E2 -24913.448} C_VEL
LIN {X 0,Y 134.361,Z 537.889,A -85,B 0,C 180,E1 -24917.925,E2 -24917.925} C_VEL
LIN {X 0,Y 133.659,Z 541.822,A -85,B 0,C 180,E1 -24922.449,E2 -24922.449} C_VEL
LIN {X 0,Y 133.466,Z 544.7,A -85,B 0,C 180,E1 -24926.984,E2 -24926.984} C_VEL
LIN {X 0,Y 133.551,Z 546.41,A -85,B 0,C 180,E1 -24930.986,E2 -24930.986} C_VEL
LIN {X 0,Y 133.548,Z 547.532,A -85,B 0,C 180,E1 -24936.044,E2 -24936.044} C_VEL
LIN {X 0,Y 133.871,Z 547.675,A -85,B 0,C 180,E1 -24939.064,E2 -24939.064} C_VEL
LIN {X 0,Y 135.238,Z 546.876,A -85,B 0,C 180,E1 -24944.495,E2 -24944.495} C_VEL
LIN {X 0,Y 135.592,Z 546.19,A -85,B 0,C 180,E1 -24946.971,E2 -24946.971} C_VEL
LIN {X 0,Y 134.946,Z 544.47,A -85,B 0,C 180,E1 -24951.097,E2 -24951.097} C_VEL
LIN {X 0,Y 134.779,Z 542.597,A -85,B 0,C 180,E1 -24954.378,E2 -24954.378} C_VEL
LIN {X 0,Y 135.686,Z 540.92,A -85,B 0,C 180,E1 -24956.747,E2 -24956.747} C_VEL
LIN {X 0,Y 136.287,Z 540.259,A -85,B 0,C 180,E1 -24957.493,E2 -24957.493} C_VEL
LIN {X 0,Y 141.347,Z 535.281,A -85,B 0,C 180,E1 -24962.1,E2 -24962.1} C_VEL
LIN {X 0,Y 146.519,Z 529.468,A -85,B 0,C 180,E1 -24965.988,E2 -24965.988} C_VEL
LIN {X 0,Y 152.193,Z 522.478,A -85,B 0,C 180,E1 -24969.418,E2 -24969.418} C_VEL
LIN {X 0,Y 158.482,Z 513.752,A -85,B 0,C 180,E1 -24972.555,E2 -24972.555} C_VEL
LIN {X 0,Y 164.1,Z 504.835,A -85,B 0,C 180,E1 -24974.965,E2 -24974.965} C_VEL
LIN {X 0,Y 169.365,Z 495.055,A -85,B 0,C 180,E1 -24977.003,E2 -24977.003} C_VEL
LIN {X 0,Y 174.271,Z 484.287,A -85,B 0,C 180,E1 -24978.688,E2 -24978.688} C_VEL
LIN {X 0,Y 178.718,Z 472.221,A -85,B 0,C 180,E1 -24980.072,E2 -24980.072} C_VEL
LIN {X 0,Y 182.135,Z 460.121,A -85,B 0,C 180,E1 -24981.087,E2 -24981.087} C_VEL
LIN {X 0,Y 184.663,Z 447.476,A -85,B 0,C 180,E1 -24981.818,E2 -24981.818} C_VEL
LIN {X 0,Y 186.366,Z 431.988,A -85,B 0,C 180,E1 -24982.368,E2 -24982.368} C_VEL
LIN {X 0,Y 187.247,Z 420.085,A -85,B 0,C 180,E1 -24982.783,E2 -24982.783} C_VEL
LIN {X 0,Y 183.518,Z 410.529,A -85,B 0,C 180,E1 -24985.404,E2 -24985.404} C_VEL
LIN {X 0,Y 179.852,Z 402.201,A -85,B 0,C 180,E1 -24988.244,E2 -24988.244} C_VEL
LIN {X 0,Y 175.856,Z 393.984,A -85,B 0,C 180,E1 -24991.77,E2 -24991.77} C_VEL
LIN {X 0,Y 172.872,Z 388.633,A -85,B 0,C 180,E1 -24994.812,E2 -24994.812} C_VEL
LIN {X 0,Y 171.001,Z 385.367,A -85,B 0,C 180,E1 -24997.018,E2 -24997.018} C_VEL
LIN {X 0,Y 168.571,Z 381.826,A -85,B 0,C 180,E1 -25000.359,E2 -25000.359} C_VEL
LIN {X 0,Y 167.982,Z 380.94,A -85,B 0,C 180,E1 -25001.318,E2 -25001.318} C_VEL
LIN {X 0,Y 165.59,Z 377.787,A -85,B 0,C 180,E1 -25006.219,E2 -25006.219} C_VEL
LIN {X 0,Y 165.049,Z 376.049,A -85,B 0,C 180,E1 -25008.182,E2 -25008.182} C_VEL
LIN {X 0,Y 164.015,Z 375.479,A -85,B 0,C 180,E1 -25015.084,E2 -25015.084} C_VEL
LIN {X 0,Y 164.887,Z 375.719,A -85,B 0,C 180,E1 -25020.611,E2 -25020.611} C_VEL
LIN {X 0,Y 165.256,Z 376.137,A -85,B 0,C 180,E1 -25021.866,E2 -25021.866} C_VEL
LIN {X 0,Y 166.877,Z 379.492,A -85,B 0,C 180,E1 -25026.12,E2 -25026.12} C_VEL
LIN {X 0,Y 168.387,Z 381.141,A -85,B 0,C 180,E1 -25028.703,E2 -25028.703} C_VEL
LIN {X 0,Y 170.697,Z 384.913,A -85,B 0,C 180,E1 -25032.031,E2 -25032.031} C_VEL
LIN {X 0,Y 171.676,Z 386.243,A -85,B 0,C 180,E1 -25033.201,E2 -25033.201} C_VEL
LIN {X 0,Y 174.85,Z 391.066,A -85,B 0,C 180,E1 -25036.567,E2 -25036.567} C_VEL
LIN {X 0,Y 178.623,Z 397.037,A -85,B 0,C 180,E1 -25039.92,E2 -25039.92} C_VEL
LIN {X 0,Y 183.705,Z 405.886,A -85,B 0,C 180,E1 -25043.76,E2 -25043.76} C_VEL
LIN {X 0,Y 186.381,Z 411.368,A -85,B 0,C 180,E1 -25045.592,E2 -25045.592} C_VEL
LIN {X 0,Y 187.719,Z 414.542,A -85,B 0,C 180,E1 -25046.479,E2 -25046.479} C_VEL
LIN {X 0,Y 185.52,Z 438.394,A -85,B 0,C 180,E1 -25047.246,E2 -25047.246} C_VEL
LIN {X 0,Y 183.047,Z 452.218,A -85,B 0,C 180,E1 -25047.983,E2 -25047.983} C_VEL
LIN {X 0,Y 179.844,Z 464.623,A -85,B 0,C 180,E1 -25049.027,E2 -25049.027} C_VEL
LIN {X 0,Y 176.085,Z 475.773,A -85,B 0,C 180,E1 -25050.33,E2 -25050.33} C_VEL
LIN {X 0,Y 171.434,Z 486.916,A -85,B 0,C 180,E1 -25052.066,E2 -25052.066} C_VEL
LIN {X 0,Y 165.878,Z 497.796,A -85,B 0,C 180,E1 -25054.289,E2 -25054.289} C_VEL
LIN {X 0,Y 160.215,Z 507.089,A -85,B 0,C 180,E1 -25056.815,E2 -25056.815} C_VEL
LIN {X 0,Y 154.862,Z 514.719,A -85,B 0,C 180,E1 -25059.509,E2 -25059.509} C_VEL
LIN {X 0,Y 148.89,Z 522.169,A -85,B 0,C 180,E1 -25062.974,E2 -25062.974} C_VEL
LIN {X 0,Y 143.568,Z 528.097,A -85,B 0,C 180,E1 -25066.736,E2 -25066.736} C_VEL
LIN {X 0,Y 138.875,Z 532.717,A -85,B 0,C 180,E1 -25070.757,E2 -25070.757} C_VEL
LIN {X 0,Y 134.898,Z 536.193,A -85,B 0,C 180,E1 -25075.032,E2 -25075.032} C_VEL
LIN {X 0,Y 132.649,Z 537.902,A -85,B 0,C 180,E1 -25078.005,E2 -25078.005} C_VEL
LIN {X 0,Y 130.744,Z 539.191,A -85,B 0,C 180,E1 -25081.065,E2 -25081.065} C_VEL
LIN {X 0,Y 129.169,Z 540.073,A -85,B 0,C 180,E1 -25084.195,E2 -25084.195} C_VEL
LIN {X 0,Y 127.253,Z 540.568,A -85,B 0,C 180,E1 -25089.868,E2 -25089.868} C_VEL
LIN {X 0,Y 126.477,Z 540.151,A -85,B 0,C 180,E1 -25093.867,E2 -25093.867} C_VEL
LIN {X 0,Y 126.099,Z 539.384,A -85,B 0,C 180,E1 -25097.116,E2 -25097.116} C_VEL
LIN {X 0,Y 126.058,Z 538.164,A -85,B 0,C 180,E1 -25100.369,E2 -25100.369} C_VEL
LIN {X 0,Y 126.763,Z 534.801,A -85,B 0,C 180,E1 -25106.354,E2 -25106.354} C_VEL
LIN {X 0,Y 127.766,Z 530.544,A -85,B 0,C 180,E1 -25111.574,E2 -25111.574} C_VEL
LIN {X 0,Y 129.415,Z 525.463,A -85,B 0,C 180,E1 -25116.233,E2 -25116.233} C_VEL
LIN {X 0,Y 131.665,Z 519.078,A -85,B 0,C 180,E1 -25120.765,E2 -25120.765} C_VEL
LIN {X 0,Y 134.699,Z 511.092,A -85,B 0,C 180,E1 -25125.12,E2 -25125.12} C_VEL
LIN {X 0,Y 137.691,Z 502.96,A -85,B 0,C 180,E1 -25128.601,E2 -25128.601} C_VEL
LIN {X 0,Y 141.257,Z 493.022,A -85,B 0,C 180,E1 -25131.908,E2 -25131.908} C_VEL
LIN {X 0,Y 144.548,Z 483.19,A -85,B 0,C 180,E1 -25134.408,E2 -25134.408} C_VEL
LIN {X 0,Y 147.781,Z 470.814,A -85,B 0,C 180,E1 -25136.856,E2 -25136.856} C_VEL
LIN {X 0,Y 150.294,Z 458.708,A -85,B 0,C 180,E1 -25138.638,E2 -25138.638} C_VEL
LIN {X 0,Y 152.226,Z 446.103,A -85,B 0,C 180,E1 -25139.944,E2 -25139.944} C_VEL
LIN {X 0,Y 153.584,Z 432.336,A -85,B 0,C 180,E1 -25140.826,E2 -25140.826} C_VEL
LIN {X 0,Y 156.43,Z 386.247,A -85,B 0,C 180,E1 -25142.695,E2 -25142.695} C_VEL
LIN {X 0,Y 152.403,Z 377.158,A -85,B 0,C 180,E1 -25144.485,E2 -25144.485} C_VEL
LIN {X 0,Y 147.075,Z 366.974,A -85,B 0,C 180,E1 -25146.964,E2 -25146.964} C_VEL
LIN {X 0,Y 140.943,Z 357,A -85,B 0,C 180,E1 -25150.066,E2 -25150.066} C_VEL
LIN {X 0,Y 137.632,Z 352.325,A -85,B 0,C 180,E1 -25151.882,E2 -25151.882} C_VEL
LIN {X 0,Y 135.394,Z 349.019,A -85,B 0,C 180,E1 -25153.212,E2 -25153.212} C_VEL
LIN {X 0,Y 133.042,Z 345.902,A -85,B 0,C 180,E1 -25154.664,E2 -25154.664} C_VEL
LIN {X 0,Y 132.278,Z 344.583,A -85,B 0,C 180,E1 -25155.183,E2 -25155.183} C_VEL
LIN {X 0,Y 130.082,Z 342.474,A -85,B 0,C 180,E1 -25156.593,E2 -25156.593} C_VEL
LIN {X 0,Y 129.09,Z 340.241,A -85,B 0,C 180,E1 -25157.379,E2 -25157.379} C_VEL
LIN {X 0,Y 128.938,Z 339.401,A -85,B 0,C 180,E1 -25157.582,E2 -25157.582} C_VEL
LIN {X 0,Y 128.919,Z 339.404,A -85,B 0,C 180,E1 -25163.153,E2 -25163.153} C_VEL
LIN {X 0,Y 128.965,Z 339.4,A -85,B 0,C 180,E1 -25166.977,E2 -25166.977} C_VEL
LIN {X 0,Y 128.995,Z 339.409,A -85,B 0,C 180,E1 -25170.654,E2 -25170.654} C_VEL
LIN {X 0,Y 129.061,Z 339.402,A -85,B 0,C 180,E1 -25177.771,E2 -25177.771} C_VEL
LIN {X 0,Y 129.137,Z 339.363,A -85,B 0,C 180,E1 -25184.209,E2 -25184.209} C_VEL
LIN {X 0,Y 129.337,Z 339.364,A -85,B 0,C 180,E1 -25187.973,E2 -25187.973} C_VEL
LIN {X 0,Y 129.454,Z 339.358,A -85,B 0,C 180,E1 -25190.626,E2 -25190.626} C_VEL
LIN {X 0,Y 130.06,Z 339.282,A -85,B 0,C 180,E1 -25199.999,E2 -25199.999} C_VEL
LIN {X 0,Y 129.463,Z 339.352,A -85,B 0,C 180,E1 -25209.372,E2 -25209.372} C_VEL
LIN {X 0,Y 129.293,Z 339.372,A -85,B 0,C 180,E1 -25212.558,E2 -25212.558} C_VEL
LIN {X 0,Y 129.108,Z 339.398,A -85,B 0,C 180,E1 -25219.063,E2 -25219.063} C_VEL
LIN {X 0,Y 129.101,Z 339.394,A -85,B 0,C 180,E1 -25222.399,E2 -25222.399} C_VEL
LIN {X 0,Y 129.02,Z 339.413,A -85,B 0,C 180,E1 -25225.834,E2 -25225.834} C_VEL
LIN {X 0,Y 129.045,Z 339.507,A -85,B 0,C 180,E1 -25231.157,E2 -25231.157} C_VEL
LIN {X 0,Y 129.834,Z 342.027,A -85,B 0,C 180,E1 -25231.855,E2 -25231.855} C_VEL
LIN {X 0,Y 131.79,Z 344.247,A -85,B 0,C 180,E1 -25233.157,E2 -25233.157} C_VEL
LIN {X 0,Y 132.693,Z 345.077,A -85,B 0,C 180,E1 -25233.716,E2 -25233.716} C_VEL
LIN {X 0,Y 134.703,Z 348.285,A -85,B 0,C 180,E1 -25235.023,E2 -25235.023} C_VEL
LIN {X 0,Y 136.239,Z 350.171,A -85,B 0,C 180,E1 -25235.929,E2 -25235.929} C_VEL
LIN {X 0,Y 139.724,Z 355.353,A -85,B 0,C 180,E1 -25237.922,E2 -25237.922} C_VEL
LIN {X 0,Y 144.43,Z 362.593,A -85,B 0,C 180,E1 -25240.375,E2 -25240.375} C_VEL
LIN {X 0,Y 149.6,Z 373.873,A -85,B 0,C 180,E1 -25243.008,E2 -25243.008} C_VEL
LIN {X 0,Y 154.075,Z 385.96,A -85,B 0,C 180,E1 -25245.209,E2 -25245.209} C_VEL
LIN {X 0,Y 155.356,Z 390.097,A -85,B 0,C 180,E1 -25245.844,E2 -25245.844} C_VEL
LIN {X 0,Y 155.861,Z 399.069,A -85,B 0,C 180,E1 -25246.516,E2 -25246.516} C_VEL
LIN {X 0,Y 152.957,Z 444.436,A -85,B 0,C 180,E1 -25248.421,E2 -25248.421} C_VEL
LIN {X 0,Y 151.279,Z 457.628,A -85,B 0,C 180,E1 -25249.431,E2 -25249.431} C_VEL
LIN {X 0,Y 148.89,Z 470.158,A -85,B 0,C 180,E1 -25250.854,E2 -25250.854} C_VEL
LIN {X 0,Y 146.146,Z 481.316,A -85,B 0,C 180,E1 -25252.621,E2 -25252.621} C_VEL
LIN {X 0,Y 142.689,Z 492.935,A -85,B 0,C 180,E1 -25255.073,E2 -25255.073} C_VEL
LIN {X 0,Y 139.226,Z 503.406,A -85,B 0,C 180,E1 -25257.995,E2 -25257.995} C_VEL
LIN {X 0,Y 135.76,Z 513.306,A -85,B 0,C 180,E1 -25261.648,E2 -25261.648} C_VEL
LIN {X 0,Y 133.167,Z 520.53,A -85,B 0,C 180,E1 -25265.029,E2 -25265.029} C_VEL
LIN {X 0,Y 130.355,Z 528.07,A -85,B 0,C 180,E1 -25269.488,E2 -25269.488} C_VEL
LIN {X 0,Y 128.262,Z 534.113,A -85,B 0,C 180,E1 -25274.102,E2 -25274.102} C_VEL
LIN {X 0,Y 127.058,Z 538.885,A -85,B 0,C 180,E1 -25278.84,E2 -25278.84} C_VEL
LIN {X 0,Y 126.469,Z 542.513,A -85,B 0,C 180,E1 -25283.621,E2 -25283.621} C_VEL
LIN {X 0,Y 126.378,Z 544.372,A -85,B 0,C 180,E1 -25286.814,E2 -25286.814} C_VEL
LIN {X 0,Y 126.503,Z 545.757,A -85,B 0,C 180,E1 -25290.002,E2 -25290.002} C_VEL
LIN {X 0,Y 126.378,Z 546.718,A -85,B 0,C 180,E1 -25293.19,E2 -25293.19} C_VEL
LIN {X 0,Y 126.859,Z 547.48,A -85,B 0,C 180,E1 -25299.569,E2 -25299.569} C_VEL
LIN {X 0,Y 128.579,Z 546.625,A -85,B 0,C 180,E1 -25305.863,E2 -25305.863} C_VEL
LIN {X 0,Y 131.769,Z 544.241,A -85,B 0,C 180,E1 -25311.925,E2 -25311.925} C_VEL
LIN {X 0,Y 135.146,Z 541.34,A -85,B 0,C 180,E1 -25316.235,E2 -25316.235} C_VEL
LIN {X 0,Y 136.287,Z 540.259,A -85,B 0,C 180,E1 -25317.493,E2 -25317.493} C_VEL
LIN {X 0,Y 137.806,Z 538.276,A -85,B 0,C 180,E1 -25319.738,E2 -25319.738} C_VEL
LIN {X 0,Y 139.014,Z 534.619,A -85,B 0,C 180,E1 -25323.533,E2 -25323.533} C_VEL
LIN {X 0,Y 140.701,Z 530.309,A -85,B 0,C 180,E1 -25327.127,E2 -25327.127} C_VEL
LIN {X 0,Y 142.88,Z 527.3,A -85,B 0,C 180,E1 -25328.983,E2 -25328.983} C_VEL
LIN {X 0,Y 148.93,Z 520.05,A -85,B 0,C 180,E1 -25332.259,E2 -25332.259} C_VEL
LIN {X 0,Y 154.489,Z 512.498,A -85,B 0,C 180,E1 -25334.842,E2 -25334.842} C_VEL
LIN {X 0,Y 160.398,Z 503.368,A -85,B 0,C 180,E1 -25337.218,E2 -25337.218} C_VEL
LIN {X 0,Y 165.853,Z 493.255,A -85,B 0,C 180,E1 -25339.242,E2 -25339.242} C_VEL
LIN {X 0,Y 170.988,Z 482.041,A -85,B 0,C 180,E1 -25340.88,E2 -25340.88} C_VEL
LIN {X 0,Y 174.947,Z 471.424,A -85,B 0,C 180,E1 -25342.036,E2 -25342.036} C_VEL
LIN {X 0,Y 178.635,Z 458.528,A -85,B 0,C 180,E1 -25343.069,E2 -25343.069} C_VEL
LIN {X 0,Y 181.146,Z 445.474,A -85,B 0,C 180,E1 -25343.77,E2 -25343.77} C_VEL
LIN {X 0,Y 183.098,Z 426.31,A -85,B 0,C 180,E1 -25344.415,E2 -25344.415} C_VEL
LIN {X 0,Y 183.312,Z 422.928,A -85,B 0,C 180,E1 -25344.559,E2 -25344.559} C_VEL
LIN {X 0,Y 179.993,Z 414.08,A -85,B 0,C 180,E1 -25347.138,E2 -25347.138} C_VEL
LIN {X 0,Y 176.1,Z 405.106,A -85,B 0,C 180,E1 -25350.487,E2 -25350.487} C_VEL
LIN {X 0,Y 173.299,Z 399.21,A -85,B 0,C 180,E1 -25353.237,E2 -25353.237} C_VEL
LIN {X 0,Y 171.046,Z 394.896,A -85,B 0,C 180,E1 -25355.74,E2 -25355.74} C_VEL
LIN {X 0,Y 169.441,Z 391.97,A -85,B 0,C 180,E1 -25357.761,E2 -25357.761} C_VEL
LIN {X 0,Y 167.065,Z 388.179,A -85,B 0,C 180,E1 -25361.311,E2 -25361.311} C_VEL
LIN {X 0,Y 164.378,Z 384.301,A -85,B 0,C 180,E1 -25367.186,E2 -25367.186} C_VEL
LIN {X 0,Y 164.072,Z 383.137,A -85,B 0,C 180,E1 -25368.469,E2 -25368.469} C_VEL
LIN {X 0,Y 163.142,Z 382.525,A -85,B 0,C 180,E1 -25375.058,E2 -25375.058} C_VEL
LIN {X 0,Y 164.014,Z 382.747,A -85,B 0,C 180,E1 -25380.614,E2 -25380.614} C_VEL
LIN {X 0,Y 164.371,Z 383.606,A -85,B 0,C 180,E1 -25381.991,E2 -25381.991} C_VEL
LIN {X 0,Y 165.993,Z 386.642,A -85,B 0,C 180,E1 -25386.153,E2 -25386.153} C_VEL
LIN {X 0,Y 167.135,Z 388.102,A -85,B 0,C 180,E1 -25388.197,E2 -25388.197} C_VEL
LIN {X 0,Y 169.515,Z 391.895,A -85,B 0,C 180,E1 -25391.737,E2 -25391.737} C_VEL
LIN {X 0,Y 173.014,Z 397.516,A -85,B 0,C 180,E1 -25395.763,E2 -25395.763} C_VEL
LIN {X 0,Y 176.482,Z 403.241,A -85,B 0,C 180,E1 -25399.03,E2 -25399.03} C_VEL
LIN {X 0,Y 181.206,Z 411.873,A -85,B 0,C 180,E1 -25402.821,E2 -25402.821} C_VEL
LIN {X 0,Y 183.456,Z 416.762,A -85,B 0,C 180,E1 -25404.47,E2 -25404.47} C_VEL
LIN {X 0,Y 183.805,Z 417.614,A -85,B 0,C 180,E1 -25404.722,E2 -25404.722} C_VEL
LIN {X 0,Y 181.622,Z 439.484,A -85,B 0,C 180,E1 -25405.422,E2 -25405.422} C_VEL
LIN {X 0,Y 179.238,Z 452.137,A -85,B 0,C 180,E1 -25406.08,E2 -25406.08} C_VEL
LIN {X 0,Y 176.114,Z 464.127,A -85,B 0,C 180,E1 -25407.074,E2 -25407.074} C_VEL
LIN {X 0,Y 172.491,Z 474.593,A -85,B 0,C 180,E1 -25408.223,E2 -25408.223} C_VEL
LIN {X 0,Y 167.842,Z 485.623,A -85,B 0,C 180,E1 -25409.883,E2 -25409.883} C_VEL
LIN {X 0,Y 162.491,Z 496.017,A -85,B 0,C 180,E1 -25411.915,E2 -25411.915} C_VEL
LIN {X 0,Y 157.101,Z 504.837,A -85,B 0,C 180,E1 -25414.144,E2 -25414.144} C_VEL
LIN {X 0,Y 151.402,Z 512.916,A -85,B 0,C 180,E1 -25416.797,E2 -25416.797} C_VEL
LIN {X 0,Y 145.04,Z 520.75,A -85,B 0,C 180,E1 -25420.253,E2 -25420.253} C_VEL
LIN {X 0,Y 140.132,Z 526.069,A -85,B 0,C 180,E1 -25423.344,E2 -25423.344} C_VEL
LIN {X 0,Y 134.866,Z 531.179,A -85,B 0,C 180,E1 -25427.353,E2 -25427.353} C_VEL
LIN {X 0,Y 130.275,Z 535.103,A -85,B 0,C 180,E1 -25431.653,E2 -25431.653} C_VEL
LIN {X 0,Y 126.156,Z 538.154,A -85,B 0,C 180,E1 -25436.683,E2 -25436.683} C_VEL
LIN {X 0,Y 122.606,Z 540.19,A -85,B 0,C 180,E1 -25442.702,E2 -25442.702} C_VEL
LIN {X 0,Y 121.209,Z 540.692,A -85,B 0,C 180,E1 -25446.051,E2 -25446.051} C_VEL
LIN {X 0,Y 120.218,Z 540.745,A -85,B 0,C 180,E1 -25449.464,E2 -25449.464} C_VEL
LIN {X 0,Y 119.498,Z 540.406,A -85,B 0,C 180,E1 -25452.896,E2 -25452.896} C_VEL
LIN {X 0,Y 119.05,Z 539.678,A -85,B 0,C 180,E1 -25456.339,E2 -25456.339} C_VEL
LIN {X 0,Y 118.962,Z 538.522,A -85,B 0,C 180,E1 -25459.789,E2 -25459.789} C_VEL
LIN {X 0,Y 119.142,Z 536.927,A -85,B 0,C 180,E1 -25463.222,E2 -25463.222} C_VEL
LIN {X 0,Y 119.818,Z 534.31,A -85,B 0,C 180,E1 -25467.551,E2 -25467.551} C_VEL
LIN {X 0,Y 120.67,Z 531.046,A -85,B 0,C 180,E1 -25471.666,E2 -25471.666} C_VEL
LIN {X 0,Y 122.368,Z 526.048,A -85,B 0,C 180,E1 -25476.593,E2 -25476.593} C_VEL
LIN {X 0,Y 124.704,Z 519.781,A -85,B 0,C 180,E1 -25481.374,E2 -25481.374} C_VEL
LIN {X 0,Y 127.86,Z 511.923,A -85,B 0,C 180,E1 -25485.949,E2 -25485.949} C_VEL
LIN {X 0,Y 131.68,Z 502.134,A -85,B 0,C 180,E1 -25490.296,E2 -25490.296} C_VEL
LIN {X 0,Y 135.51,Z 491.913,A -85,B 0,C 180,E1 -25493.697,E2 -25493.697} C_VEL
LIN {X 0,Y 138.955,Z 481.758,A -85,B 0,C 180,E1 -25496.264,E2 -25496.264} C_VEL
LIN {X 0,Y 141.951,Z 470.743,A -85,B 0,C 180,E1 -25498.457,E2 -25498.457} C_VEL
LIN {X 0,Y 144.605,Z 458.555,A -85,B 0,C 180,E1 -25500.278,E2 -25500.278} C_VEL
LIN {X 0,Y 146.628,Z 445.737,A -85,B 0,C 180,E1 -25501.615,E2 -25501.615} C_VEL
LIN {X 0,Y 147.96,Z 432.665,A -85,B 0,C 180,E1 -25502.467,E2 -25502.467} C_VEL
LIN {X 0,Y 150.879,Z 388.263,A -85,B 0,C 180,E1 -25504.295,E2 -25504.295} C_VEL
LIN {X 0,Y 145.278,Z 376.193,A -85,B 0,C 180,E1 -25507.012,E2 -25507.012} C_VEL
LIN {X 0,Y 139.287,Z 365.565,A -85,B 0,C 180,E1 -25510.147,E2 -25510.147} C_VEL
LIN {X 0,Y 134.251,Z 357.909,A -85,B 0,C 180,E1 -25513.059,E2 -25513.059} C_VEL
LIN {X 0,Y 131.72,Z 354.265,A -85,B 0,C 180,E1 -25514.656,E2 -25514.656} C_VEL
LIN {X 0,Y 128.933,Z 350.34,A -85,B 0,C 180,E1 -25516.548,E2 -25516.548} C_VEL
LIN {X 0,Y 126.465,Z 347.291,A -85,B 0,C 180,E1 -25518.326,E2 -25518.326} C_VEL
LIN {X 0,Y 125.574,Z 345.66,A -85,B 0,C 180,E1 -25519.057,E2 -25519.057} C_VEL
LIN {X 0,Y 123.081,Z 343.512,A -85,B 0,C 180,E1 -25520.979,E2 -25520.979} C_VEL
LIN {X 0,Y 122.017,Z 341.226,A -85,B 0,C 180,E1 -25522.005,E2 -25522.005} C_VEL
LIN {X 0,Y 121.86,Z 340.289,A -85,B 0,C 180,E1 -25522.384,E2 -25522.384} C_VEL
LIN {X 0,Y 121.902,Z 340.269,A -85,B 0,C 180,E1 -25524.792,E2 -25524.792} C_VEL
LIN {X 0,Y 121.911,Z 340.296,A -85,B 0,C 180,E1 -25529.846,E2 -25529.846} C_VEL
LIN {X 0,Y 121.973,Z 340.277,A -85,B 0,C 180,E1 -25537.199,E2 -25537.199} C_VEL
